LIN {X 0,Y 199.177,Z 547.457,A -85,B 0,C 180,E1 21373.917,E2 21373.917} C_VEL
LIN {X 0,Y 215.115,Z 524.972,A -85,B 0,C 180,E1 21379.948,E2 21379.948} C_VEL
LIN {X 0,Y 227.752,Z 503.08,A -85,B 0,C 180,E1 21383.961,E2 21383.961} C_VEL
LIN {X 0,Y 227.913,Z 485.066,A -85,B 0,C 180,E1 21390.32,E2 21390.32} C_VEL
LIN {X 0,Y 225.682,Z 468.338,A -85,B 0,C 180,E1 21397.834,E2 21397.834} C_VEL
LIN {X 0,Y 223.444,Z 458.289,A -85,B 0,C 180,E1 21404.278,E2 21404.278} C_VEL
LIN {X 0,Y 222.036,Z 452.317,A -85,B 0,C 180,E1 21410.188,E2 21410.188} C_VEL
LIN {X 0,Y 221.908,Z 448.763,A -85,B 0,C 180,E1 21416.091,E2 21416.091} C_VEL
LIN {X 0,Y 222.152,Z 448.898,A -85,B 0,C 180,E1 21420.003,E2 21420.003} C_VEL
LIN {X 0,Y 223.226,Z 453.842,A -85,B 0,C 180,E1 21426.819,E2 21426.819} C_VEL
LIN {X 0,Y 226.174,Z 464.487,A -85,B 0,C 180,E1 21434.54,E2 21434.54} C_VEL
LIN {X 0,Y 229.513,Z 478.492,A -85,B 0,C 180,E1 21441.276,E2 21441.276} C_VEL
LIN {X 0,Y 231.824,Z 496.438,A -85,B 0,C 180,E1 21447.624,E2 21447.624} C_VEL
LIN {X 0,Y 231.749,Z 502.452,A -85,B 0,C 180,E1 21449.308,E2 21449.308} C_VEL
LIN {X 0,Y 215.555,Z 532.804,A -85,B 0,C 180,E1 21453.677,E2 21453.677} C_VEL
LIN {X 0,Y 197.818,Z 560.36,A -85,B 0,C 180,E1 21460.055,E2 21460.055} C_VEL
LIN {X 0,Y 181.866,Z 582.088,A -85,B 0,C 180,E1 21468.235,E2 21468.235} C_VEL
LIN {X 0,Y 169.045,Z 599.486,A -85,B 0,C 180,E1 21478.996,E2 21478.996} C_VEL
LIN {X 0,Y 162.169,Z 610.738,A -85,B 0,C 180,E1 21490.92,E2 21490.92} C_VEL
LIN {X 0,Y 160.605,Z 615.153,A -85,B 0,C 180,E1 21499.125,E2 21499.125} C_VEL
LIN {X 0,Y 160.77,Z 617.402,A -85,B 0,C 180,E1 21509.992,E2 21509.992} C_VEL
LIN {X 0,Y 160.648,Z 615.185,A -85,B 0,C 180,E1 21520.856,E2 21520.856} C_VEL
LIN {X 0,Y 161.483,Z 612.541,A -85,B 0,C 180,E1 21526.327,E2 21526.327} C_VEL
LIN {X 0,Y 170.904,Z 608.235,A -85,B 0,C 180,E1 21542.098,E2 21542.098} C_VEL
LIN {X 0,Y 192.339,Z 598.523,A -85,B 0,C 180,E1 21555.096,E2 21555.096} C_VEL
LIN {X 0,Y 202.815,Z 593.917,A -85,B 0,C 180,E1 21558.952,E2 21558.952} C_VEL
LIN {X 0,Y 200.293,Z 594.401,A -85,B 0,C 180,E1 21560.543,E2 21560.543} C_VEL
LIN {X 0,Y 180.77,Z 597.692,A -85,B 0,C 180,E1 21569.832,E2 21569.832} C_VEL
LIN {X 0,Y 169.639,Z 596.938,A -85,B 0,C 180,E1 21579.082,E2 21579.082} C_VEL
LIN {X 0,Y 162.377,Z 590.884,A -85,B 0,C 180,E1 21591.957,E2 21591.957} C_VEL
LIN {X 0,Y 160.932,Z 581.155,A -85,B 0,C 180,E1 21602.692,E2 21602.692} C_VEL
LIN {X 0,Y 162.1,Z 567.404,A -85,B 0,C 180,E1 21612.606,E2 21612.606} C_VEL
LIN {X 0,Y 165.856,Z 547.555,A -85,B 0,C 180,E1 21622.423,E2 21622.423} C_VEL
LIN {X 0,Y 167.025,Z 542.957,A -85,B 0,C 180,E1 21624.287,E2 21624.287} C_VEL
LIN {X 0,Y 181.526,Z 540.142,A -85,B 0,C 180,E1 21632.822,E2 21632.822} C_VEL
LIN {X 0,Y 209.455,Z 532.398,A -85,B 0,C 180,E1 21641.296,E2 21641.296} C_VEL
LIN {X 0,Y 209.889,Z 533.058,A -85,B 0,C 180,E1 21641.79,E2 21641.79} C_VEL
LIN {X 0,Y 192.98,Z 555.356,A -85,B 0,C 180,E1 21648.886,E2 21648.886} C_VEL
LIN {X 0,Y 182.434,Z 564.426,A -85,B 0,C 180,E1 21652.185,E2 21652.185} C_VEL
LIN {X 0,Y 172.325,Z 572.215,A -85,B 0,C 180,E1 21656.038,E2 21656.038} C_VEL
LIN {X 0,Y 160.406,Z 584.48,A -85,B 0,C 180,E1 21667.828,E2 21667.828} C_VEL
LIN {X 0,Y 155.075,Z 590.148,A -85,B 0,C 180,E1 21678.749,E2 21678.749} C_VEL
LIN {X 0,Y 153.359,Z 591.986,A -85,B 0,C 180,E1 21690.008,E2 21690.008} C_VEL
LIN {X 0,Y 156.005,Z 589.027,A -85,B 0,C 180,E1 21703.985,E2 21703.985} C_VEL
LIN {X 0,Y 163.582,Z 581.161,A -85,B 0,C 180,E1 21716.088,E2 21716.088} C_VEL
LIN {X 0,Y 176.711,Z 567.47,A -85,B 0,C 180,E1 21726.858,E2 21726.858} C_VEL
LIN {X 0,Y 193.582,Z 548.12,A -85,B 0,C 180,E1 21735.541,E2 21735.541} C_VEL
LIN {X 0,Y 211.371,Z 523.809,A -85,B 0,C 180,E1 21741.996,E2 21741.996} C_VEL
LIN {X 0,Y 221.798,Z 506.936,A -85,B 0,C 180,E1 21745.004,E2 21745.004} C_VEL
LIN {X 0,Y 222.86,Z 490.693,A -85,B 0,C 180,E1 21750.937,E2 21750.937} C_VEL
LIN {X 0,Y 221.632,Z 475.531,A -85,B 0,C 180,E1 21757.936,E2 21757.936} C_VEL
LIN {X 0,Y 219.974,Z 465.484,A -85,B 0,C 180,E1 21764.499,E2 21764.499} C_VEL
LIN {X 0,Y 218.806,Z 459.156,A -85,B 0,C 180,E1 21771.173,E2 21771.173} C_VEL
LIN {X 0,Y 218.997,Z 456.251,A -85,B 0,C 180,E1 21776.039,E2 21776.039} C_VEL
LIN {X 0,Y 219.233,Z 456.387,A -85,B 0,C 180,E1 21780.003,E2 21780.003} C_VEL
LIN {X 0,Y 220.349,Z 462.641,A -85,B 0,C 180,E1 21787.901,E2 21787.901} C_VEL
LIN {X 0,Y 223.108,Z 474.069,A -85,B 0,C 180,E1 21795.752,E2 21795.752} C_VEL
LIN {X 0,Y 225.619,Z 489.59,A -85,B 0,C 180,E1 21802.7,E2 21802.7} C_VEL
LIN {X 0,Y 226.479,Z 503.724,A -85,B 0,C 180,E1 21807.631,E2 21807.631} C_VEL
LIN {X 0,Y 209.961,Z 534.007,A -85,B 0,C 180,E1 21812.2,E2 21812.2} C_VEL
LIN {X 0,Y 191.432,Z 561.307,A -85,B 0,C 180,E1 21818.711,E2 21818.711} C_VEL
LIN {X 0,Y 174.369,Z 583.318,A -85,B 0,C 180,E1 21827.422,E2 21827.422} C_VEL
LIN {X 0,Y 160.676,Z 600.703,A -85,B 0,C 180,E1 21839.171,E2 21839.171} C_VEL
LIN {X 0,Y 154.488,Z 610.163,A -85,B 0,C 180,E1 21850.074,E2 21850.074} C_VEL
LIN {X 0,Y 152.751,Z 614.505,A -85,B 0,C 180,E1 21858.558,E2 21858.558} C_VEL
LIN {X 0,Y 152.874,Z 616.764,A -85,B 0,C 180,E1 21869.992,E2 21869.992} C_VEL
LIN {X 0,Y 152.815,Z 614.539,A -85,B 0,C 180,E1 21881.42,E2 21881.42} C_VEL
LIN {X 0,Y 153.758,Z 611.875,A -85,B 0,C 180,E1 21887.172,E2 21887.172} C_VEL
LIN {X 0,Y 166.907,Z 606.908,A -85,B 0,C 180,E1 21905.966,E2 21905.966} C_VEL
LIN {X 0,Y 192.972,Z 596.975,A -85,B 0,C 180,E1 21919.08,E2 21919.08} C_VEL
LIN {X 0,Y 190.683,Z 597.243,A -85,B 0,C 180,E1 21920.565,E2 21920.565} C_VEL
LIN {X 0,Y 167.495,Z 598.655,A -85,B 0,C 180,E1 21933.129,E2 21933.129} C_VEL
LIN {X 0,Y 156.735,Z 594.166,A -85,B 0,C 180,E1 21946.023,E2 21946.023} C_VEL
LIN {X 0,Y 153.33,Z 584.856,A -85,B 0,C 180,E1 21958.582,E2 21958.582} C_VEL
LIN {X 0,Y 153.787,Z 570.942,A -85,B 0,C 180,E1 21970.171,E2 21970.171} C_VEL
LIN {X 0,Y 157.168,Z 550.928,A -85,B 0,C 180,E1 21981.171,E2 21981.171} C_VEL
LIN {X 0,Y 157.889,Z 548.939,A -85,B 0,C 180,E1 21982.549,E2 21982.549} C_VEL
LIN {X 0,Y 176.43,Z 545.25,A -85,B 0,C 180,E1 21993.896,E2 21993.896} C_VEL
LIN {X 0,Y 200.361,Z 539.066,A -85,B 0,C 180,E1 22001.377,E2 22001.377} C_VEL
LIN {X 0,Y 185.688,Z 557.62,A -85,B 0,C 180,E1 22007.987,E2 22007.987} C_VEL
LIN {X 0,Y 172.325,Z 572.215,A -85,B 0,C 180,E1 22016.038,E2 22016.038} C_VEL
LIN {X 0,Y 162.691,Z 578.921,A -85,B 0,C 180,E1 22020.5,E2 22020.5} C_VEL
LIN {X 0,Y 153.884,Z 584.343,A -85,B 0,C 180,E1 22025.631,E2 22025.631} C_VEL
LIN {X 0,Y 147.346,Z 590.785,A -85,B 0,C 180,E1 22038.151,E2 22038.151} C_VEL
LIN {X 0,Y 145.513,Z 592.621,A -85,B 0,C 180,E1 22050.009,E2 22050.009} C_VEL
LIN {X 0,Y 148.359,Z 589.665,A -85,B 0,C 180,E1 22064.721,E2 22064.721} C_VEL
LIN {X 0,Y 156.51,Z 581.805,A -85,B 0,C 180,E1 22077.362,E2 22077.362} C_VEL
LIN {X 0,Y 170.435,Z 568.125,A -85,B 0,C 180,E1 22088.457,E2 22088.457} C_VEL
LIN {X 0,Y 188.147,Z 548.795,A -85,B 0,C 180,E1 22097.254,E2 22097.254} C_VEL
LIN {X 0,Y 206.616,Z 524.515,A -85,B 0,C 180,E1 22103.717,E2 22103.717} C_VEL
LIN {X 0,Y 216.312,Z 509.416,A -85,B 0,C 180,E1 22106.433,E2 22106.433} C_VEL
LIN {X 0,Y 217.663,Z 493.427,A -85,B 0,C 180,E1 22112.765,E2 22112.765} C_VEL
LIN {X 0,Y 217.088,Z 479.857,A -85,B 0,C 180,E1 22119.596,E2 22119.596} C_VEL
LIN {X 0,Y 215.907,Z 470.26,A -85,B 0,C 180,E1 22126.727,E2 22126.727} C_VEL
LIN {X 0,Y 215.801,Z 463.629,A -85,B 0,C 180,E1 22135.98,E2 22135.98} C_VEL
LIN {X 0,Y 216.058,Z 463.769,A -85,B 0,C 180,E1 22140.003,E2 22140.003} C_VEL
LIN {X 0,Y 217.033,Z 470.12,A -85,B 0,C 180,E1 22148.022,E2 22148.022} C_VEL
LIN {X 0,Y 219.239,Z 482.003,A -85,B 0,C 180,E1 22156.037,E2 22156.037} C_VEL
LIN {X 0,Y 220.857,Z 498.201,A -85,B 0,C 180,E1 22163.215,E2 22163.215} C_VEL
LIN {X 0,Y 220.919,Z 507.282,A -85,B 0,C 180,E1 22166.459,E2 22166.459} C_VEL
LIN {X 0,Y 203.853,Z 536.285,A -85,B 0,C 180,E1 22170.849,E2 22170.849} C_VEL
LIN {X 0,Y 185.494,Z 561.798,A -85,B 0,C 180,E1 22177.13,E2 22177.13} C_VEL
LIN {X 0,Y 168.145,Z 582.98,A -85,B 0,C 180,E1 22185.713,E2 22185.713} C_VEL
LIN {X 0,Y 153.562,Z 600.243,A -85,B 0,C 180,E1 22197.81,E2 22197.81} C_VEL
LIN {X 0,Y 146.69,Z 609.895,A -85,B 0,C 180,E1 22209.67,E2 22209.67} C_VEL
LIN {X 0,Y 144.904,Z 613.856,A -85,B 0,C 180,E1 22217.93,E2 22217.93} C_VEL
LIN {X 0,Y 144.977,Z 616.125,A -85,B 0,C 180,E1 22229.991,E2 22229.991} C_VEL
LIN {X 0,Y 144.97,Z 613.892,A -85,B 0,C 180,E1 22242.047,E2 22242.047} C_VEL
LIN {X 0,Y 146.908,Z 610.149,A -85,B 0,C 180,E1 22250.483,E2 22250.483} C_VEL
LIN {X 0,Y 160.601,Z 606.569,A -85,B 0,C 180,E1 22267.777,E2 22267.777} C_VEL
LIN {X 0,Y 182.654,Z 599.585,A -85,B 0,C 180,E1 22279.069,E2 22279.069} C_VEL
LIN {X 0,Y 181.918,Z 599.433,A -85,B 0,C 180,E1 22280.198,E2 22280.198} C_VEL
LIN {X 0,Y 160.523,Z 599.431,A -85,B 0,C 180,E1 22291.861,E2 22291.861} C_VEL
LIN {X 0,Y 148.97,Z 594.046,A -85,B 0,C 180,E1 22305.479,E2 22305.479} C_VEL
LIN {X 0,Y 145.459,Z 584.242,A -85,B 0,C 180,E1 22318.505,E2 22318.505} C_VEL
LIN {X 0,Y 145.985,Z 569.601,A -85,B 0,C 180,E1 22330.721,E2 22330.721} C_VEL
LIN {X 0,Y 148.737,Z 554.448,A -85,B 0,C 180,E1 22340.088,E2 22340.088} C_VEL
LIN {X 0,Y 171.246,Z 550.073,A -85,B 0,C 180,E1 22355.07,E2 22355.07} C_VEL
LIN {X 0,Y 190.552,Z 545.467,A -85,B 0,C 180,E1 22361.307,E2 22361.307} C_VEL
LIN {X 0,Y 175.103,Z 563.43,A -85,B 0,C 180,E1 22368.767,E2 22368.767} C_VEL
LIN {X 0,Y 160.002,Z 578.515,A -85,B 0,C 180,E1 22379.091,E2 22379.091} C_VEL
LIN {X 0,Y 153.884,Z 584.343,A -85,B 0,C 180,E1 22385.631,E2 22385.631} C_VEL
LIN {X 0,Y 146.298,Z 588.632,A -85,B 0,C 180,E1 22391.428,E2 22391.428} C_VEL
LIN {X 0,Y 139.489,Z 591.502,A -85,B 0,C 180,E1 22397.847,E2 22397.847} C_VEL
LIN {X 0,Y 137.636,Z 593.258,A -85,B 0,C 180,E1 22410.009,E2 22410.009} C_VEL
LIN {X 0,Y 140.642,Z 590.392,A -85,B 0,C 180,E1 22425.301,E2 22425.301} C_VEL
LIN {X 0,Y 149.53,Z 582.448,A -85,B 0,C 180,E1 22438.755,E2 22438.755} C_VEL
LIN {X 0,Y 164.301,Z 568.777,A -85,B 0,C 180,E1 22450.176,E2 22450.176} C_VEL
LIN {X 0,Y 182.875,Z 549.472,A -85,B 0,C 180,E1 22459.072,E2 22459.072} C_VEL
LIN {X 0,Y 202.045,Z 525.224,A -85,B 0,C 180,E1 22465.522,E2 22465.522} C_VEL
LIN {X 0,Y 210.882,Z 512.011,A -85,B 0,C 180,E1 22467.927,E2 22467.927} C_VEL
LIN {X 0,Y 212.565,Z 497.474,A -85,B 0,C 180,E1 22474.12,E2 22474.12} C_VEL
LIN {X 0,Y 212.641,Z 484.92,A -85,B 0,C 180,E1 22480.892,E2 22480.892} C_VEL
LIN {X 0,Y 212.092,Z 475.095,A -85,B 0,C 180,E1 22489.148,E2 22489.148} C_VEL
LIN {X 0,Y 212.433,Z 470.784,A -85,B 0,C 180,E1 22496.226,E2 22496.226} C_VEL
LIN {X 0,Y 212.665,Z 471.048,A -85,B 0,C 180,E1 22500.003,E2 22500.003} C_VEL
LIN {X 0,Y 213.404,Z 477.484,A -85,B 0,C 180,E1 22508.159,E2 22508.159} C_VEL
LIN {X 0,Y 214.836,Z 488.174,A -85,B 0,C 180,E1 22515.448,E2 22515.448} C_VEL
LIN {X 0,Y 215.654,Z 503.707,A -85,B 0,C 180,E1 22522.581,E2 22522.581} C_VEL
LIN {X 0,Y 214.959,Z 511.066,A -85,B 0,C 180,E1 22525.103,E2 22525.103} C_VEL
LIN {X 0,Y 196.7,Z 539.99,A -85,B 0,C 180,E1 22529.744,E2 22529.744} C_VEL
LIN {X 0,Y 176.998,Z 565.69,A -85,B 0,C 180,E1 22536.573,E2 22536.573} C_VEL
LIN {X 0,Y 158.766,Z 586.294,A -85,B 0,C 180,E1 22545.972,E2 22545.972} C_VEL
LIN {X 0,Y 144.748,Z 601.89,A -85,B 0,C 180,E1 22558.459,E2 22558.459} C_VEL
LIN {X 0,Y 138.364,Z 610.501,A -85,B 0,C 180,E1 22570.828,E2 22570.828} C_VEL
LIN {X 0,Y 136.72,Z 614.84,A -85,B 0,C 180,E1 22583.633,E2 22583.633} C_VEL
LIN {X 0,Y 137.078,Z 615.485,A -85,B 0,C 180,E1 22589.991,E2 22589.991} C_VEL
LIN {X 0,Y 137.141,Z 613.244,A -85,B 0,C 180,E1 22602.745,E2 22602.745} C_VEL
LIN {X 0,Y 140.214,Z 608.914,A -85,B 0,C 180,E1 22613.505,E2 22613.505} C_VEL
LIN {X 0,Y 158.032,Z 605.249,A -85,B 0,C 180,E1 22632.102,E2 22632.102} C_VEL
LIN {X 0,Y 171.29,Z 601.783,A -85,B 0,C 180,E1 22638.657,E2 22638.657} C_VEL
LIN {X 0,Y 172.797,Z 601.214,A -85,B 0,C 180,E1 22639.877,E2 22639.877} C_VEL
LIN {X 0,Y 153.627,Z 600.092,A -85,B 0,C 180,E1 22650.476,E2 22650.476} C_VEL
LIN {X 0,Y 140.769,Z 593.255,A -85,B 0,C 180,E1 22665.839,E2 22665.839} C_VEL
LIN {X 0,Y 137.429,Z 581.903,A -85,B 0,C 180,E1 22679.996,E2 22679.996} C_VEL
LIN {X 0,Y 138.221,Z 568.205,A -85,B 0,C 180,E1 22691.304,E2 22691.304} C_VEL
LIN {X 0,Y 139.695,Z 559.704,A -85,B 0,C 180,E1 22697.335,E2 22697.335} C_VEL
LIN {X 0,Y 161.307,Z 555.607,A -85,B 0,C 180,E1 22714.267,E2 22714.267} C_VEL
LIN {X 0,Y 180.578,Z 551.515,A -85,B 0,C 180,E1 22721.239,E2 22721.239} C_VEL
LIN {X 0,Y 177.835,Z 555.21,A -85,B 0,C 180,E1 22722.92,E2 22722.92} C_VEL
LIN {X 0,Y 160.43,Z 572.578,A -85,B 0,C 180,E1 22732.176,E2 22732.176} C_VEL
LIN {X 0,Y 146.442,Z 585.224,A -85,B 0,C 180,E1 22744.702,E2 22744.702} C_VEL
LIN {X 0,Y 139.489,Z 591.502,A -85,B 0,C 180,E1 22757.847,E2 22757.847} C_VEL
LIN {X 0,Y 133.921,Z 593.276,A -85,B 0,C 180,E1 22764.753,E2 22764.753} C_VEL
LIN {X 0,Y 129.705,Z 593.729,A -85,B 0,C 180,E1 22772.169,E2 22772.169} C_VEL
LIN {X 0,Y 133.161,Z 590.92,A -85,B 0,C 180,E1 22786.523,E2 22786.523} C_VEL
LIN {X 0,Y 142.641,Z 583.091,A -85,B 0,C 180,E1 22800.285,E2 22800.285} C_VEL
LIN {X 0,Y 158.347,Z 569.428,A -85,B 0,C 180,E1 22812.021,E2 22812.021} C_VEL
LIN {X 0,Y 177.792,Z 550.149,A -85,B 0,C 180,E1 22820.999,E2 22820.999} C_VEL
LIN {X 0,Y 197.697,Z 525.933,A -85,B 0,C 180,E1 22827.402,E2 22827.402} C_VEL
LIN {X 0,Y 205.54,Z 514.4,A -85,B 0,C 180,E1 22829.642,E2 22829.642} C_VEL
LIN {X 0,Y 207.567,Z 501.324,A -85,B 0,C 180,E1 22835.594,E2 22835.594} C_VEL
LIN {X 0,Y 208.143,Z 490.302,A -85,B 0,C 180,E1 22841.997,E2 22841.997} C_VEL
LIN {X 0,Y 208.188,Z 481.816,A -85,B 0,C 180,E1 22849.528,E2 22849.528} C_VEL
LIN {X 0,Y 208.744,Z 478.088,A -85,B 0,C 180,E1 22855.844,E2 22855.844} C_VEL
LIN {X 0,Y 209.065,Z 478.207,A -85,B 0,C 180,E1 22860.003,E2 22860.003} C_VEL
LIN {X 0,Y 209.479,Z 484.8,A -85,B 0,C 180,E1 22868.313,E2 22868.313} C_VEL
LIN {X 0,Y 210.352,Z 495.679,A -85,B 0,C 180,E1 22875.66,E2 22875.66} C_VEL
LIN {X 0,Y 210.201,Z 511.241,A -85,B 0,C 180,E1 22882.779,E2 22882.779} C_VEL
LIN {X 0,Y 209.033,Z 514.658,A -85,B 0,C 180,E1 22883.673,E2 22883.673} C_VEL
LIN {X 0,Y 189.597,Z 543.646,A -85,B 0,C 180,E1 22888.542,E2 22888.542} C_VEL
LIN {X 0,Y 169.651,Z 567.882,A -85,B 0,C 180,E1 22895.446,E2 22895.446} C_VEL
LIN {X 0,Y 150.704,Z 587.978,A -85,B 0,C 180,E1 22905.303,E2 22905.303} C_VEL
LIN {X 0,Y 136.66,Z 602.512,A -85,B 0,C 180,E1 22918.239,E2 22918.239} C_VEL
LIN {X 0,Y 129.844,Z 611.31,A -85,B 0,C 180,E1 22933.042,E2 22933.042} C_VEL
LIN {X 0,Y 128.808,Z 614.195,A -85,B 0,C 180,E1 22943.24,E2 22943.24} C_VEL
LIN {X 0,Y 129.204,Z 614.848,A -85,B 0,C 180,E1 22949.99,E2 22949.99} C_VEL
LIN {X 0,Y 129.329,Z 612.596,A -85,B 0,C 180,E1 22963.529,E2 22963.529} C_VEL
LIN {X 0,Y 132.998,Z 607.618,A -85,B 0,C 180,E1 22975.033,E2 22975.033} C_VEL
LIN {X 0,Y 152.158,Z 604.861,A -85,B 0,C 180,E1 22994.134,E2 22994.134} C_VEL
LIN {X 0,Y 162.831,Z 602.613,A -85,B 0,C 180,E1 22999.392,E2 22999.392} C_VEL
LIN {X 0,Y 140.546,Z 598.526,A -85,B 0,C 180,E1 23014.473,E2 23014.473} C_VEL
LIN {X 0,Y 131.264,Z 589.48,A -85,B 0,C 180,E1 23030.033,E2 23030.033} C_VEL
LIN {X 0,Y 129.471,Z 577.442,A -85,B 0,C 180,E1 23043.347,E2 23043.347} C_VEL
LIN {X 0,Y 130.723,Z 564.733,A -85,B 0,C 180,E1 23053.388,E2 23053.388} C_VEL
LIN {X 0,Y 155.911,Z 559.992,A -85,B 0,C 180,E1 23075.629,E2 23075.629} C_VEL
LIN {X 0,Y 170.564,Z 557.157,A -85,B 0,C 180,E1 23081.17,E2 23081.17} C_VEL
LIN {X 0,Y 169.026,Z 559.373,A -85,B 0,C 180,E1 23082.491,E2 23082.491} C_VEL
LIN {X 0,Y 150.549,Z 576.474,A -85,B 0,C 180,E1 23092.9,E2 23092.9} C_VEL
LIN {X 0,Y 138.702,Z 586.399,A -85,B 0,C 180,E1 23104.123,E2 23104.123} C_VEL
LIN {X 0,Y 131.729,Z 592.174,A -85,B 0,C 180,E1 23117.29,E2 23117.29} C_VEL
LIN {X 0,Y 129.705,Z 593.729,A -85,B 0,C 180,E1 23132.169,E2 23132.169} C_VEL
LIN {X 0,Y 128.791,Z 593.589,A -85,B 0,C 180,E1 23136.027,E2 23136.027} C_VEL
LIN {X 0,Y 125.412,Z 591.794,A -85,B 0,C 180,E1 23146.863,E2 23146.863} C_VEL
LIN {X 0,Y 125.743,Z 591.444,A -85,B 0,C 180,E1 23147.846,E2 23147.846} C_VEL
LIN {X 0,Y 137.412,Z 582.478,A -85,B 0,C 180,E1 23163.438,E2 23163.438} C_VEL
LIN {X 0,Y 154.74,Z 568.203,A -85,B 0,C 180,E1 23175.191,E2 23175.191} C_VEL
LIN {X 0,Y 174.256,Z 549.401,A -85,B 0,C 180,E1 23183.491,E2 23183.491} C_VEL
LIN {X 0,Y 194.63,Z 525.25,A -85,B 0,C 180,E1 23189.649,E2 23189.649} C_VEL
LIN {X 0,Y 199.715,Z 518.278,A -85,B 0,C 180,E1 23190.894,E2 23190.894} C_VEL
LIN {X 0,Y 202.28,Z 507.251,A -85,B 0,C 180,E1 23196.031,E2 23196.031} C_VEL
LIN {X 0,Y 203.544,Z 496.214,A -85,B 0,C 180,E1 23202.695,E2 23202.695} C_VEL
LIN {X 0,Y 204.115,Z 488.415,A -85,B 0,C 180,E1 23209.962,E2 23209.962} C_VEL
LIN {X 0,Y 204.853,Z 485.115,A -85,B 0,C 180,E1 23215.765,E2 23215.765} C_VEL
LIN {X 0,Y 205.181,Z 485.204,A -85,B 0,C 180,E1 23220.003,E2 23220.003} C_VEL
LIN {X 0,Y 205.276,Z 490.817,A -85,B 0,C 180,E1 23227.418,E2 23227.418} C_VEL
LIN {X 0,Y 205.573,Z 501.41,A -85,B 0,C 180,E1 23234.942,E2 23234.942} C_VEL
LIN {X 0,Y 204.756,Z 515.453,A -85,B 0,C 180,E1 23241.699,E2 23241.699} C_VEL
LIN {X 0,Y 184.073,Z 545.131,A -85,B 0,C 180,E1 23246.834,E2 23246.834} C_VEL
LIN {X 0,Y 162.766,Z 569.644,A -85,B 0,C 180,E1 23254.057,E2 23254.057} C_VEL
LIN {X 0,Y 142.99,Z 589.205,A -85,B 0,C 180,E1 23264.371,E2 23264.371} C_VEL
LIN {X 0,Y 128.55,Z 603.092,A -85,B 0,C 180,E1 23277.985,E2 23277.985} C_VEL
LIN {X 0,Y 122.174,Z 610.659,A -85,B 0,C 180,E1 23291.942,E2 23291.942} C_VEL
LIN {X 0,Y 120.899,Z 613.55,A -85,B 0,C 180,E1 23302.796,E2 23302.796} C_VEL
LIN {X 0,Y 121.14,Z 614.157,A -85,B 0,C 180,E1 23310.976,E2 23310.976} C_VEL
LIN {X 0,Y 121.548,Z 611.947,A -85,B 0,C 180,E1 23324.414,E2 23324.414} C_VEL
LIN {X 0,Y 126.873,Z 606.301,A -85,B 0,C 180,E1 23338.498,E2 23338.498} C_VEL
LIN {X 0,Y 146.519,Z 604.336,A -85,B 0,C 180,E1 23356.314,E2 23356.314} C_VEL
LIN {X 0,Y 152.448,Z 603.18,A -85,B 0,C 180,E1 23359.793,E2 23359.793} C_VEL
LIN {X 0,Y 133.459,Z 598.549,A -85,B 0,C 180,E1 23373.011,E2 23373.011} C_VEL
LIN {X 0,Y 123.623,Z 588.993,A -85,B 0,C 180,E1 23389.117,E2 23389.117} C_VEL
LIN {X 0,Y 121.644,Z 577.998,A -85,B 0,C 180,E1 23401.766,E2 23401.766} C_VEL
LIN {X 0,Y 122.248,Z 569.693,A -85,B 0,C 180,E1 23409.799,E2 23409.799} C_VEL
LIN {X 0,Y 150.501,Z 564.18,A -85,B 0,C 180,E1 23437.12,E2 23437.12} C_VEL
LIN {X 0,Y 160.838,Z 562.349,A -85,B 0,C 180,E1 23441.21,E2 23441.21} C_VEL
LIN {X 0,Y 156.837,Z 566.466,A -85,B 0,C 180,E1 23443.654,E2 23443.654} C_VEL
LIN {X 0,Y 139.17,Z 581.176,A -85,B 0,C 180,E1 23454.907,E2 23454.907} C_VEL
LIN {X 0,Y 127.249,Z 590.356,A -85,B 0,C 180,E1 23469.1,E2 23469.1} C_VEL
LIN {X 0,Y 122.336,Z 594.051,A -85,B 0,C 180,E1 23482.902,E2 23482.902} C_VEL
LIN {X 0,Y 122.363,Z 594.017,A -85,B 0,C 180,E1 23497.118,E2 23497.118} C_VEL
LIN {X 0,Y 125.743,Z 591.444,A -85,B 0,C 180,E1 23507.846,E2 23507.846} C_VEL
LIN {X 0,Y 126.247,Z 588.646,A -85,B 0,C 180,E1 23515.709,E2 23515.709} C_VEL
LIN {X 0,Y 128.708,Z 584.718,A -85,B 0,C 180,E1 23523.345,E2 23523.345} C_VEL
LIN {X 0,Y 146.969,Z 570.732,A -85,B 0,C 180,E1 23536.156,E2 23536.156} C_VEL
LIN {X 0,Y 168.311,Z 551.494,A -85,B 0,C 180,E1 23545.176,E2 23545.176} C_VEL
LIN {X 0,Y 189.679,Z 527.345,A -85,B 0,C 180,E1 23551.413,E2 23551.413} C_VEL
LIN {X 0,Y 194.77,Z 520.67,A -85,B 0,C 180,E1 23552.63,E2 23552.63} C_VEL
LIN {X 0,Y 197.791,Z 508.325,A -85,B 0,C 180,E1 23559.204,E2 23559.204} C_VEL
LIN {X 0,Y 199.196,Z 499.247,A -85,B 0,C 180,E1 23565.739,E2 23565.739} C_VEL
LIN {X 0,Y 199.973,Z 494.357,A -85,B 0,C 180,E1 23571.294,E2 23571.294} C_VEL
LIN {X 0,Y 200.695,Z 491.986,A -85,B 0,C 180,E1 23575.677,E2 23575.677} C_VEL
LIN {X 0,Y 201.068,Z 492.055,A -85,B 0,C 180,E1 23580.003,E2 23580.003} C_VEL
LIN {X 0,Y 200.949,Z 497.876,A -85,B 0,C 180,E1 23587.579,E2 23587.579} C_VEL
LIN {X 0,Y 200.666,Z 507.493,A -85,B 0,C 180,E1 23594.476,E2 23594.476} C_VEL
LIN {X 0,Y 199.104,Z 519.316,A -85,B 0,C 180,E1 23600.285,E2 23600.285} C_VEL
LIN {X 0,Y 178.301,Z 547.105,A -85,B 0,C 180,E1 23605.125,E2 23605.125} C_VEL
LIN {X 0,Y 156.437,Z 570.883,A -85,B 0,C 180,E1 23612.366,E2 23612.366} C_VEL
LIN {X 0,Y 135.315,Z 590.374,A -85,B 0,C 180,E1 23623.331,E2 23623.331} C_VEL
LIN {X 0,Y 120.473,Z 603.668,A -85,B 0,C 180,E1 23637.706,E2 23637.706} C_VEL
LIN {X 0,Y 113.714,Z 611.259,A -85,B 0,C 180,E1 23654.546,E2 23654.546} C_VEL
LIN {X 0,Y 113.431,Z 613.572,A -85,B 0,C 180,E1 23669.989,E2 23669.989} C_VEL
LIN {X 0,Y 113.786,Z 611.298,A -85,B 0,C 180,E1 23685.421,E2 23685.421} C_VEL
LIN {X 0,Y 121.122,Z 604.822,A -85,B 0,C 180,E1 23702.075,E2 23702.075} C_VEL
LIN {X 0,Y 141.104,Z 603.54,A -85,B 0,C 180,E1 23718.667,E2 23718.667} C_VEL
LIN {X 0,Y 142.023,Z 603.118,A -85,B 0,C 180,E1 23720.235,E2 23720.235} C_VEL
LIN {X 0,Y 123.495,Z 596.805,A -85,B 0,C 180,E1 23734.587,E2 23734.587} C_VEL
LIN {X 0,Y 114.825,Z 585.036,A -85,B 0,C 180,E1 23752.419,E2 23752.419} C_VEL
LIN {X 0,Y 113.823,Z 574.715,A -85,B 0,C 180,E1 23763.782,E2 23763.782} C_VEL
LIN {X 0,Y 148.775,Z 567.469,A -85,B 0,C 180,E1 23800.305,E2 23800.305} C_VEL
LIN {X 0,Y 150.456,Z 567.18,A -85,B 0,C 180,E1 23800.96,E2 23800.96} C_VEL
LIN {X 0,Y 149.132,Z 569.101,A -85,B 0,C 180,E1 23802.64,E2 23802.64} C_VEL
LIN {X 0,Y 130.769,Z 583.28,A -85,B 0,C 180,E1 23814.642,E2 23814.642} C_VEL
LIN {X 0,Y 119.894,Z 590.996,A -85,B 0,C 180,E1 23827.751,E2 23827.751} C_VEL
LIN {X 0,Y 114.533,Z 594.687,A -85,B 0,C 180,E1 23842.416,E2 23842.416} C_VEL
LIN {X 0,Y 114.56,Z 594.654,A -85,B 0,C 180,E1 23857.605,E2 23857.605} C_VEL
LIN {X 0,Y 119.939,Z 590.902,A -85,B 0,C 180,E1 23872.263,E2 23872.263} C_VEL
LIN {X 0,Y 128.708,Z 584.718,A -85,B 0,C 180,E1 23883.345,E2 23883.345} C_VEL
LIN {X 0,Y 132.962,Z 579.725,A -85,B 0,C 180,E1 23890.477,E2 23890.477} C_VEL
LIN {X 0,Y 138.748,Z 573.608,A -85,B 0,C 180,E1 23896.984,E2 23896.984} C_VEL
LIN {X 0,Y 161.131,Z 554.747,A -85,B 0,C 180,E1 23906.52,E2 23906.52} C_VEL
LIN {X 0,Y 182.659,Z 532.195,A -85,B 0,C 180,E1 23912.74,E2 23912.74} C_VEL
LIN {X 0,Y 189.708,Z 523.378,A -85,B 0,C 180,E1 23914.455,E2 23914.455} C_VEL
LIN {X 0,Y 193.301,Z 510.949,A -85,B 0,C 180,E1 23921.746,E2 23921.746} C_VEL
LIN {X 0,Y 194.901,Z 503.458,A -85,B 0,C 180,E1 23928.182,E2 23928.182} C_VEL
LIN {X 0,Y 196.319,Z 498.748,A -85,B 0,C 180,E1 23935.58,E2 23935.58} C_VEL
LIN {X 0,Y 196.748,Z 498.793,A -85,B 0,C 180,E1 23940.003,E2 23940.003} C_VEL
LIN {X 0,Y 196.276,Z 504.821,A -85,B 0,C 180,E1 23947.76,E2 23947.76} C_VEL
LIN {X 0,Y 195.363,Z 514.44,A -85,B 0,C 180,E1 23954.59,E2 23954.59} C_VEL
LIN {X 0,Y 194.339,Z 521.071,A -85,B 0,C 180,E1 23958.159,E2 23958.159} C_VEL
LIN {X 0,Y 182.411,Z 537.524,A -85,B 0,C 180,E1 23960.961,E2 23960.961} C_VEL
LIN {X 0,Y 159.54,Z 563.045,A -85,B 0,C 180,E1 23967.156,E2 23967.156} C_VEL
LIN {X 0,Y 136.783,Z 583.896,A -85,B 0,C 180,E1 23976.621,E2 23976.621} C_VEL
LIN {X 0,Y 118.051,Z 599.351,A -85,B 0,C 180,E1 23990.312,E2 23990.312} C_VEL
LIN {X 0,Y 108.316,Z 607.874,A -85,B 0,C 180,E1 24005.196,E2 24005.196} C_VEL
LIN {X 0,Y 105.103,Z 612.26,A -85,B 0,C 180,E1 24021.706,E2 24021.706} C_VEL
LIN {X 0,Y 105.521,Z 612.932,A -85,B 0,C 180,E1 24029.988,E2 24029.988} C_VEL
LIN {X 0,Y 106.06,Z 610.649,A -85,B 0,C 180,E1 24046.575,E2 24046.575} C_VEL
LIN {X 0,Y 114.459,Z 603.224,A -85,B 0,C 180,E1 24064.19,E2 24064.19} C_VEL
LIN {X 0,Y 131.203,Z 602.977,A -85,B 0,C 180,E1 24078.577,E2 24078.577} C_VEL
LIN {X 0,Y 132.476,Z 602.664,A -85,B 0,C 180,E1 24080.064,E2 24080.064} C_VEL
LIN {X 0,Y 112.457,Z 593.218,A -85,B 0,C 180,E1 24098.266,E2 24098.266} C_VEL
LIN {X 0,Y 106.232,Z 579.517,A -85,B 0,C 180,E1 24117.953,E2 24117.953} C_VEL
LIN {X 0,Y 141.459,Z 571.618,A -85,B 0,C 180,E1 24161.496,E2 24161.496} C_VEL
LIN {X 0,Y 122.614,Z 585.15,A -85,B 0,C 180,E1 24174.105,E2 24174.105} C_VEL
LIN {X 0,Y 110.578,Z 592.913,A -85,B 0,C 180,E1 24189.997,E2 24189.997} C_VEL
LIN {X 0,Y 106.161,Z 595.805,A -85,B 0,C 180,E1 24210.012,E2 24210.012} C_VEL
LIN {X 0,Y 110.658,Z 592.837,A -85,B 0,C 180,E1 24230.013,E2 24230.013} C_VEL
LIN {X 0,Y 122.717,Z 585.018,A -85,B 0,C 180,E1 24245.887,E2 24245.887} C_VEL
LIN {X 0,Y 138.748,Z 573.608,A -85,B 0,C 180,E1 24256.984,E2 24256.984} C_VEL
LIN {X 0,Y 145.791,Z 566.543,A -85,B 0,C 180,E1 24262.806,E2 24262.806} C_VEL
LIN {X 0,Y 153.721,Z 558.273,A -85,B 0,C 180,E1 24267.879,E2 24267.879} C_VEL
LIN {X 0,Y 176.359,Z 536.014,A -85,B 0,C 180,E1 24274.31,E2 24274.31} C_VEL
LIN {X 0,Y 184.875,Z 525.825,A -85,B 0,C 180,E1 24276.53,E2 24276.53} C_VEL
LIN {X 0,Y 188.21,Z 516.071,A -85,B 0,C 180,E1 24282.723,E2 24282.723} C_VEL
LIN {X 0,Y 190.065,Z 509.68,A -85,B 0,C 180,E1 24288.517,E2 24288.517} C_VEL
LIN {X 0,Y 191.729,Z 505.39,A -85,B 0,C 180,E1 24295.474,E2 24295.474} C_VEL
LIN {X 0,Y 192.242,Z 505.382,A -85,B 0,C 180,E1 24300.003,E2 24300.003} C_VEL
LIN {X 0,Y 191.517,Z 510.375,A -85,B 0,C 180,E1 24306.813,E2 24306.813} C_VEL
LIN {X 0,Y 190.084,Z 519.74,A -85,B 0,C 180,E1 24313.827,E2 24313.827} C_VEL
LIN {X 0,Y 188.764,Z 525.25,A -85,B 0,C 180,E1 24316.758,E2 24316.758} C_VEL
LIN {X 0,Y 166.131,Z 552.093,A -85,B 0,C 180,E1 24321.679,E2 24321.679} C_VEL
LIN {X 0,Y 141.851,Z 575.224,A -85,B 0,C 180,E1 24329.456,E2 24329.456} C_VEL
LIN {X 0,Y 120.113,Z 592.498,A -85,B 0,C 180,E1 24340.848,E2 24340.848} C_VEL
LIN {X 0,Y 104.291,Z 604.464,A -85,B 0,C 180,E1 24357.004,E2 24357.004} C_VEL
LIN {X 0,Y 98.294,Z 609.957,A -85,B 0,C 180,E1 24372.045,E2 24372.045} C_VEL
LIN {X 0,Y 97.605,Z 612.292,A -85,B 0,C 180,E1 24389.987,E2 24389.987} C_VEL
LIN {X 0,Y 98.385,Z 609.999,A -85,B 0,C 180,E1 24407.91,E2 24407.91} C_VEL
LIN {X 0,Y 109.588,Z 601.533,A -85,B 0,C 180,E1 24428.423,E2 24428.423} C_VEL
LIN {X 0,Y 121.353,Z 601.851,A -85,B 0,C 180,E1 24438.447,E2 24438.447} C_VEL
LIN {X 0,Y 122.254,Z 601.481,A -85,B 0,C 180,E1 24440.295,E2 24440.295} C_VEL
LIN {X 0,Y 104.061,Z 591.15,A -85,B 0,C 180,E1 24458.666,E2 24458.666} C_VEL
LIN {X 0,Y 99.646,Z 584.49,A -85,B 0,C 180,E1 24469.817,E2 24469.817} C_VEL
LIN {X 0,Y 103.957,Z 579.95,A -85,B 0,C 180,E1 24496.927,E2 24496.927} C_VEL
LIN {X 0,Y 130.166,Z 575.774,A -85,B 0,C 180,E1 24520.557,E2 24520.557} C_VEL
LIN {X 0,Y 131.081,Z 576.037,A -85,B 0,C 180,E1 24521.707,E2 24521.707} C_VEL
LIN {X 0,Y 112.663,Z 587.997,A -85,B 0,C 180,E1 24535.225,E2 24535.225} C_VEL
LIN {X 0,Y 101.458,Z 594.611,A -85,B 0,C 180,E1 24552.65,E2 24552.65} C_VEL
LIN {X 0,Y 98.304,Z 596.441,A -85,B 0,C 180,E1 24570.013,E2 24570.013} C_VEL
LIN {X 0,Y 103.258,Z 593.477,A -85,B 0,C 180,E1 24591.516,E2 24591.516} C_VEL
LIN {X 0,Y 116.38,Z 585.661,A -85,B 0,C 180,E1 24608.177,E2 24608.177} C_VEL
LIN {X 0,Y 136.479,Z 572.038,A -85,B 0,C 180,E1 24620.956,E2 24620.956} C_VEL
LIN {X 0,Y 153.721,Z 558.273,A -85,B 0,C 180,E1 24627.879,E2 24627.879} C_VEL
LIN {X 0,Y 162.316,Z 549.148,A -85,B 0,C 180,E1 24632.342,E2 24632.342} C_VEL
LIN {X 0,Y 169.739,Z 540.345,A -85,B 0,C 180,E1 24635.859,E2 24635.859} C_VEL
LIN {X 0,Y 171.051,Z 538.908,A -85,B 0,C 180,E1 24636.196,E2 24636.196} C_VEL
LIN {X 0,Y 179.579,Z 529.464,A -85,B 0,C 180,E1 24638.044,E2 24638.044} C_VEL
LIN {X 0,Y 183.541,Z 519.915,A -85,B 0,C 180,E1 24644.734,E2 24644.734} C_VEL
LIN {X 0,Y 185.756,Z 513.907,A -85,B 0,C 180,E1 24651.472,E2 24651.472} C_VEL
LIN {X 0,Y 186.899,Z 511.864,A -85,B 0,C 180,E1 24655.357,E2 24655.357} C_VEL
LIN {X 0,Y 187.452,Z 511.783,A -85,B 0,C 180,E1 24660.003,E2 24660.003} C_VEL
LIN {X 0,Y 186.336,Z 517.407,A -85,B 0,C 180,E1 24667.337,E2 24667.337} C_VEL
LIN {X 0,Y 184.501,Z 525.76,A -85,B 0,C 180,E1 24673.542,E2 24673.542} C_VEL
LIN {X 0,Y 183.51,Z 528.397,A -85,B 0,C 180,E1 24674.907,E2 24674.907} C_VEL
LIN {X 0,Y 159.169,Z 555.612,A -85,B 0,C 180,E1 24680.049,E2 24680.049} C_VEL
LIN {X 0,Y 133.326,Z 578.257,A -85,B 0,C 180,E1 24688.335,E2 24688.335} C_VEL
LIN {X 0,Y 110.372,Z 595.026,A -85,B 0,C 180,E1 24701.008,E2 24701.008} C_VEL
LIN {X 0,Y 96.191,Z 604.826,A -85,B 0,C 180,E1 24716.558,E2 24716.558} C_VEL
LIN {X 0,Y 90.687,Z 609.307,A -85,B 0,C 180,E1 24730.481,E2 24730.481} C_VEL
LIN {X 0,Y 89.686,Z 611.651,A -85,B 0,C 180,E1 24749.986,E2 24749.986} C_VEL
LIN {X 0,Y 90.782,Z 609.351,A -85,B 0,C 180,E1 24769.468,E2 24769.468} C_VEL
LIN {X 0,Y 103.394,Z 600.651,A -85,B 0,C 180,E1 24791.2,E2 24791.2} C_VEL
LIN {X 0,Y 108.277,Z 599.951,A -85,B 0,C 180,E1 24795.639,E2 24795.639} C_VEL
LIN {X 0,Y 112.601,Z 600.18,A -85,B 0,C 180,E1 24798.957,E2 24798.957} C_VEL
LIN {X 0,Y 110.396,Z 598.904,A -85,B 0,C 180,E1 24801.888,E2 24801.888} C_VEL
LIN {X 0,Y 95.564,Z 589.617,A -85,B 0,C 180,E1 24819.112,E2 24819.112} C_VEL
LIN {X 0,Y 93.303,Z 584.487,A -85,B 0,C 180,E1 24849.332,E2 24849.332} C_VEL
LIN {X 0,Y 121.327,Z 579.691,A -85,B 0,C 180,E1 24881.539,E2 24881.539} C_VEL
LIN {X 0,Y 104.51,Z 589.598,A -85,B 0,C 180,E1 24894.604,E2 24894.604} C_VEL
LIN {X 0,Y 93.947,Z 595.25,A -85,B 0,C 180,E1 24911.213,E2 24911.213} C_VEL
LIN {X 0,Y 90.44,Z 597.077,A -85,B 0,C 180,E1 24930.014,E2 24930.014} C_VEL
LIN {X 0,Y 95.952,Z 594.116,A -85,B 0,C 180,E1 24953.246,E2 24953.246} C_VEL
LIN {X 0,Y 110.034,Z 586.423,A -85,B 0,C 180,E1 24970.542,E2 24970.542} C_VEL
LIN {X 0,Y 131.632,Z 572.69,A -85,B 0,C 180,E1 24983.635,E2 24983.635} C_VEL
LIN {X 0,Y 156.013,Z 553.498,A -85,B 0,C 180,E1 24992.328,E2 24992.328} C_VEL
LIN {X 0,Y 171.051,Z 538.908,A -85,B 0,C 180,E1 24996.196,E2 24996.196} C_VEL
LIN {X 0,Y 174.504,Z 534.139,A -85,B 0,C 180,E1 24998.248,E2 24998.248} C_VEL
LIN {X 0,Y 176.733,Z 528.402,A -85,B 0,C 180,E1 25002.946,E2 25002.946} C_VEL
LIN {X 0,Y 179.659,Z 522.115,A -85,B 0,C 180,E1 25008.673,E2 25008.673} C_VEL
LIN {X 0,Y 181.806,Z 518.152,A -85,B 0,C 180,E1 25015.227,E2 25015.227} C_VEL
LIN {X 0,Y 182.435,Z 518.05,A -85,B 0,C 180,E1 25020.003,E2 25020.003} C_VEL
LIN {X 0,Y 181.346,Z 522.497,A -85,B 0,C 180,E1 25026.164,E2 25026.164} C_VEL
LIN {X 0,Y 179.052,Z 530.432,A -85,B 0,C 180,E1 25032.501,E2 25032.501} C_VEL
LIN {X 0,Y 172.819,Z 538.065,A -85,B 0,C 180,E1 25033.952,E2 25033.952} C_VEL
LIN {X 0,Y 146.737,Z 563.766,A -85,B 0,C 180,E1 25039.677,E2 25039.677} C_VEL
LIN {X 0,Y 120.9,Z 583.925,A -85,B 0,C 180,E1 25048.749,E2 25048.749} C_VEL
LIN {X 0,Y 97.825,Z 598.94,A -85,B 0,C 180,E1 25063.712,E2 25063.712} C_VEL
LIN {X 0,Y 84.738,Z 607.35,A -85,B 0,C 180,E1 25083.304,E2 25083.304} C_VEL
LIN {X 0,Y 81.482,Z 610.322,A -85,B 0,C 180,E1 25099.276,E2 25099.276} C_VEL
LIN {X 0,Y 81.765,Z 611.01,A -85,B 0,C 180,E1 25109.984,E2 25109.984} C_VEL
LIN {X 0,Y 83.245,Z 608.701,A -85,B 0,C 180,E1 25131.313,E2 25131.313} C_VEL
LIN {X 0,Y 97.389,Z 600.04,A -85,B 0,C 180,E1 25154.232,E2 25154.232} C_VEL
LIN {X 0,Y 101.928,Z 597.878,A -85,B 0,C 180,E1 25157.938,E2 25157.938} C_VEL
LIN {X 0,Y 103.252,Z 597.744,A -85,B 0,C 180,E1 25160.01,E2 25160.01} C_VEL
LIN {X 0,Y 95.99,Z 594.702,A -85,B 0,C 180,E1 25166.488,E2 25166.488} C_VEL
LIN {X 0,Y 84.352,Z 588.846,A -85,B 0,C 180,E1 25199.993,E2 25199.993} C_VEL
LIN {X 0,Y 110.316,Z 583.083,A -85,B 0,C 180,E1 25240.198,E2 25240.198} C_VEL
LIN {X 0,Y 111.172,Z 583.313,A -85,B 0,C 180,E1 25241.594,E2 25241.594} C_VEL
LIN {X 0,Y 91.407,Z 593.554,A -85,B 0,C 180,E1 25260.223,E2 25260.223} C_VEL
LIN {X 0,Y 83.453,Z 597.231,A -85,B 0,C 180,E1 25279.564,E2 25279.564} C_VEL
LIN {X 0,Y 83.455,Z 597.203,A -85,B 0,C 180,E1 25300.467,E2 25300.467} C_VEL
LIN {X 0,Y 91.459,Z 593.465,A -85,B 0,C 180,E1 25319.791,E2 25319.791} C_VEL
LIN {X 0,Y 111.362,Z 583.11,A -85,B 0,C 180,E1 25338.409,E2 25338.409} C_VEL
LIN {X 0,Y 135.782,Z 567.306,A -85,B 0,C 180,E1 25349.87,E2 25349.87} C_VEL
LIN {X 0,Y 160.427,Z 547.043,A -85,B 0,C 180,E1 25356.961,E2 25356.961} C_VEL
LIN {X 0,Y 174.736,Z 532.454,A -85,B 0,C 180,E1 25360.075,E2 25360.075} C_VEL
LIN {X 0,Y 176.733,Z 528.402,A -85,B 0,C 180,E1 25362.946,E2 25362.946} C_VEL
LIN {X 0,Y 177.335,Z 525.849,A -85,B 0,C 180,E1 25366.361,E2 25366.361} C_VEL
LIN {X 0,Y 176.218,Z 524.646,A -85,B 0,C 180,E1 25374.411,E2 25374.411} C_VEL
LIN {X 0,Y 177.237,Z 524.161,A -85,B 0,C 180,E1 25380.003,E2 25380.003} C_VEL
LIN {X 0,Y 175.379,Z 529.961,A -85,B 0,C 180,E1 25387.443,E2 25387.443} C_VEL
LIN {X 0,Y 173.98,Z 533.897,A -85,B 0,C 180,E1 25390.659,E2 25390.659} C_VEL
LIN {X 0,Y 149.239,Z 558.745,A -85,B 0,C 180,E1 25395.45,E2 25395.45} C_VEL
LIN {X 0,Y 121.752,Z 580.186,A -85,B 0,C 180,E1 25403.475,E2 25403.475} C_VEL
LIN {X 0,Y 97.902,Z 595.13,A -85,B 0,C 180,E1 25415.701,E2 25415.701} C_VEL
LIN {X 0,Y 80.01,Z 605.24,A -85,B 0,C 180,E1 25435.394,E2 25435.394} C_VEL
LIN {X 0,Y 73.656,Z 609.677,A -85,B 0,C 180,E1 25458.121,E2 25458.121} C_VEL
LIN {X 0,Y 73.858,Z 610.37,A -85,B 0,C 180,E1 25469.982,E2 25469.982} C_VEL
LIN {X 0,Y 75.8,Z 608.05,A -85,B 0,C 180,E1 25493.525,E2 25493.525} C_VEL
LIN {X 0,Y 90.753,Z 599.956,A -85,B 0,C 180,E1 25516.818,E2 25516.818} C_VEL
LIN {X 0,Y 93.947,Z 598.103,A -85,B 0,C 180,E1 25519.858,E2 25519.858} C_VEL
LIN {X 0,Y 76.904,Z 591.508,A -85,B 0,C 180,E1 25559.993,E2 25559.993} C_VEL
LIN {X 0,Y 97.849,Z 586.605,A -85,B 0,C 180,E1 25598.227,E2 25598.227} C_VEL
LIN {X 0,Y 101.1,Z 586.496,A -85,B 0,C 180,E1 25601.539,E2 25601.539} C_VEL
LIN {X 0,Y 84.621,Z 594.196,A -85,B 0,C 180,E1 25617.557,E2 25617.557} C_VEL
LIN {X 0,Y 75.723,Z 597.868,A -85,B 0,C 180,E1 25638.485,E2 25638.485} C_VEL
LIN {X 0,Y 75.729,Z 597.839,A -85,B 0,C 180,E1 25661.549,E2 25661.549} C_VEL
LIN {X 0,Y 84.679,Z 594.106,A -85,B 0,C 180,E1 25682.454,E2 25682.454} C_VEL
LIN {X 0,Y 103.695,Z 585.063,A -85,B 0,C 180,E1 25700.059,E2 25700.059} C_VEL
LIN {X 0,Y 128.902,Z 570.102,A -85,B 0,C 180,E1 25711.795,E2 25711.795} C_VEL
LIN {X 0,Y 154.195,Z 550.602,A -85,B 0,C 180,E1 25718.889,E2 25718.889} C_VEL
LIN {X 0,Y 169.717,Z 535.804,A -85,B 0,C 180,E1 25722.041,E2 25722.041} C_VEL
LIN {X 0,Y 173.44,Z 529.347,A -85,B 0,C 180,E1 25727.412,E2 25727.412} C_VEL
LIN {X 0,Y 176.218,Z 524.646,A -85,B 0,C 180,E1 25734.411,E2 25734.411} C_VEL
LIN {X 0,Y 175.77,Z 525.349,A -85,B 0,C 180,E1 25737.922,E2 25737.922} C_VEL
LIN {X 0,Y 170.257,Z 534.05,A -85,B 0,C 180,E1 25745.588,E2 25745.588} C_VEL
LIN {X 0,Y 168.543,Z 537.822,A -85,B 0,C 180,E1 25748.81,E2 25748.81} C_VEL
LIN {X 0,Y 141.825,Z 562.6,A -85,B 0,C 180,E1 25753.543,E2 25753.543} C_VEL
LIN {X 0,Y 113.936,Z 582.573,A -85,B 0,C 180,E1 25761.514,E2 25761.514} C_VEL
LIN {X 0,Y 87.598,Z 597.487,A -85,B 0,C 180,E1 25775.744,E2 25775.744} C_VEL
LIN {X 0,Y 70.898,Z 605.905,A -85,B 0,C 180,E1 25796.812,E2 25796.812} C_VEL
LIN {X 0,Y 65.837,Z 609.028,A -85,B 0,C 180,E1 25816.686,E2 25816.686} C_VEL
LIN {X 0,Y 65.927,Z 609.729,A -85,B 0,C 180,E1 25829.98,E2 25829.98} C_VEL
LIN {X 0,Y 68.492,Z 607.399,A -85,B 0,C 180,E1 25856.215,E2 25856.215} C_VEL
LIN {X 0,Y 81.911,Z 600.946,A -85,B 0,C 180,E1 25877.649,E2 25877.649} C_VEL
LIN {X 0,Y 83.632,Z 599.585,A -85,B 0,C 180,E1 25880.902,E2 25880.902} C_VEL
LIN {X 0,Y 69.368,Z 593.951,A -85,B 0,C 180,E1 25919.992,E2 25919.992} C_VEL
LIN {X 0,Y 90.826,Z 589.209,A -85,B 0,C 180,E1 25960.224,E2 25960.224} C_VEL
LIN {X 0,Y 89.705,Z 590.009,A -85,B 0,C 180,E1 25962.45,E2 25962.45} C_VEL
LIN {X 0,Y 71.932,Z 597.163,A -85,B 0,C 180,E1 25985.126,E2 25985.126} C_VEL
LIN {X 0,Y 66.815,Z 598.988,A -85,B 0,C 180,E1 26010.019,E2 26010.019} C_VEL
LIN {X 0,Y 71.998,Z 597.111,A -85,B 0,C 180,E1 26034.889,E2 26034.889} C_VEL
LIN {X 0,Y 90.385,Z 589.624,A -85,B 0,C 180,E1 26057.943,E2 26057.943} C_VEL
LIN {X 0,Y 116.06,Z 576.515,A -85,B 0,C 180,E1 26071.726,E2 26071.726} C_VEL
LIN {X 0,Y 143.172,Z 558.084,A -85,B 0,C 180,E1 26079.82,E2 26079.82} C_VEL
LIN {X 0,Y 164.725,Z 539.221,A -85,B 0,C 180,E1 26084.132,E2 26084.132} C_VEL
LIN {X 0,Y 168.765,Z 533.313,A -85,B 0,C 180,E1 26089.668,E2 26089.668} C_VEL
LIN {X 0,Y 170.976,Z 530.334,A -85,B 0,C 180,E1 26094.923,E2 26094.923} C_VEL
LIN {X 0,Y 171.837,Z 530.136,A -85,B 0,C 180,E1 26100.003,E2 26100.003} C_VEL
LIN {X 0,Y 170.257,Z 534.05,A -85,B 0,C 180,E1 26105.588,E2 26105.588} C_VEL
LIN {X 0,Y 167.011,Z 538.168,A -85,B 0,C 180,E1 26107.058,E2 26107.058} C_VEL
LIN {X 0,Y 154.112,Z 550.092,A -85,B 0,C 180,E1 26107.926,E2 26107.926} C_VEL
LIN {X 0,Y 126.437,Z 572.132,A -85,B 0,C 180,E1 26113.333,E2 26113.333} C_VEL
LIN {X 0,Y 98.395,Z 589.165,A -85,B 0,C 180,E1 26122.572,E2 26122.572} C_VEL
LIN {X 0,Y 73.588,Z 601.161,A -85,B 0,C 180,E1 26139.484,E2 26139.484} C_VEL
LIN {X 0,Y 61.219,Z 606.696,A -85,B 0,C 180,E1 26160.332,E2 26160.332} C_VEL
LIN {X 0,Y 57.992,Z 609.087,A -85,B 0,C 180,E1 26189.978,E2 26189.978} C_VEL
LIN {X 0,Y 61.384,Z 606.75,A -85,B 0,C 180,E1 26219.531,E2 26219.531} C_VEL
LIN {X 0,Y 73.992,Z 601.44,A -85,B 0,C 180,E1 26239.588,E2 26239.588} C_VEL
LIN {X 0,Y 73.594,Z 600.832,A -85,B 0,C 180,E1 26241.883,E2 26241.883} C_VEL
LIN {X 0,Y 61.766,Z 596.17,A -85,B 0,C 180,E1 26279.991,E2 26279.991} C_VEL
LIN {X 0,Y 76.638,Z 592.508,A -85,B 0,C 180,E1 26316.334,E2 26316.334} C_VEL
LIN {X 0,Y 80.789,Z 592.16,A -85,B 0,C 180,E1 26321.471,E2 26321.471} C_VEL
LIN {X 0,Y 64.838,Z 597.802,A -85,B 0,C 180,E1 26342.184,E2 26342.184} C_VEL
LIN {X 0,Y 58.949,Z 599.625,A -85,B 0,C 180,E1 26370.022,E2 26370.022} C_VEL
LIN {X 0,Y 64.907,Z 597.751,A -85,B 0,C 180,E1 26397.829,E2 26397.829} C_VEL
LIN {X 0,Y 85.288,Z 590.267,A -85,B 0,C 180,E1 26421.892,E2 26421.892} C_VEL
LIN {X 0,Y 112.522,Z 577.164,A -85,B 0,C 180,E1 26435.283,E2 26435.283} C_VEL
LIN {X 0,Y 140.652,Z 558.749,A -85,B 0,C 180,E1 26442.83,E2 26442.83} C_VEL
LIN {X 0,Y 159.76,Z 542.788,A -85,B 0,C 180,E1 26446.336,E2 26446.336} C_VEL
LIN {X 0,Y 162.524,Z 539.383,A -85,B 0,C 180,E1 26449.267,E2 26449.267} C_VEL
LIN {X 0,Y 165.259,Z 536.158,A -85,B 0,C 180,E1 26454.747,E2 26454.747} C_VEL
LIN {X 0,Y 166.191,Z 535.869,A -85,B 0,C 180,E1 26460.003,E2 26460.003} C_VEL
LIN {X 0,Y 164.157,Z 540.222,A -85,B 0,C 180,E1 26465.967,E2 26465.967} C_VEL
LIN {X 0,Y 160.69,Z 543.926,A -85,B 0,C 180,E1 26466.956,E2 26466.956} C_VEL
LIN {X 0,Y 154.112,Z 550.092,A -85,B 0,C 180,E1 26467.926,E2 26467.926} C_VEL
LIN {X 0,Y 140.333,Z 560.926,A -85,B 0,C 180,E1 26468.537,E2 26468.537} C_VEL
LIN {X 0,Y 125.969,Z 570.63,A -85,B 0,C 180,E1 26469.429,E2 26469.429} C_VEL
LIN {X 0,Y 95.55,Z 588.497,A -85,B 0,C 180,E1 26478.029,E2 26478.029} C_VEL
LIN {X 0,Y 68.694,Z 600.499,A -85,B 0,C 180,E1 26494.231,E2 26494.231} C_VEL
LIN {X 0,Y 53.842,Z 606.228,A -85,B 0,C 180,E1 26517.534,E2 26517.534} C_VEL
LIN {X 0,Y 50.05,Z 608.444,A -85,B 0,C 180,E1 26549.974,E2 26549.974} C_VEL
LIN {X 0,Y 54.545,Z 606.101,A -85,B 0,C 180,E1 26583.69,E2 26583.69} C_VEL
LIN {X 0,Y 62.004,Z 603.391,A -85,B 0,C 180,E1 26597.066,E2 26597.066} C_VEL
LIN {X 0,Y 64.18,Z 602.026,A -85,B 0,C 180,E1 26602.3,E2 26602.3} C_VEL
LIN {X 0,Y 56.645,Z 596.777,A -85,B 0,C 180,E1 26655.491,E2 26655.491} C_VEL
LIN {X 0,Y 70.573,Z 594.468,A -85,B 0,C 180,E1 26680.047,E2 26680.047} C_VEL
LIN {X 0,Y 57.972,Z 598.44,A -85,B 0,C 180,E1 26698.54,E2 26698.54} C_VEL
LIN {X 0,Y 51.072,Z 600.262,A -85,B 0,C 180,E1 26730.025,E2 26730.025} C_VEL
LIN {X 0,Y 58.043,Z 598.389,A -85,B 0,C 180,E1 26761.47,E2 26761.47} C_VEL
LIN {X 0,Y 80.858,Z 590.829,A -85,B 0,C 180,E1 26786.457,E2 26786.457} C_VEL
LIN {X 0,Y 109.451,Z 577.811,A -85,B 0,C 180,E1 26799.046,E2 26799.046} C_VEL
LIN {X 0,Y 138.522,Z 559.419,A -85,B 0,C 180,E1 26805.96,E2 26805.96} C_VEL
LIN {X 0,Y 155.737,Z 545.523,A -85,B 0,C 180,E1 26808.793,E2 26808.793} C_VEL
LIN {X 0,Y 159.225,Z 541.803,A -85,B 0,C 180,E1 26814.548,E2 26814.548} C_VEL
LIN {X 0,Y 160.336,Z 541.439,A -85,B 0,C 180,E1 26820.004,E2 26820.004} C_VEL
LIN {X 0,Y 158.971,Z 543.996,A -85,B 0,C 180,E1 26823.885,E2 26823.885} C_VEL
LIN {X 0,Y 131.957,Z 566.445,A -85,B 0,C 180,E1 26828.228,E2 26828.228} C_VEL
LIN {X 0,Y 125.969,Z 570.63,A -85,B 0,C 180,E1 26829.429,E2 26829.429} C_VEL
LIN {X 0,Y 110.99,Z 579.364,A -85,B 0,C 180,E1 26830.718,E2 26830.718} C_VEL
LIN {X 0,Y 95.462,Z 586.813,A -85,B 0,C 180,E1 26832.568,E2 26832.568} C_VEL
LIN {X 0,Y 65.006,Z 599.634,A -85,B 0,C 180,E1 26847.77,E2 26847.77} C_VEL
LIN {X 0,Y 47.813,Z 605.385,A -85,B 0,C 180,E1 26870.673,E2 26870.673} C_VEL
LIN {X 0,Y 42.12,Z 607.802,A -85,B 0,C 180,E1 26909.969,E2 26909.969} C_VEL
LIN {X 0,Y 48.049,Z 605.451,A -85,B 0,C 180,E1 26949.027,E2 26949.027} C_VEL
LIN {X 0,Y 53.655,Z 603.724,A -85,B 0,C 180,E1 26959.014,E2 26959.014} C_VEL
LIN {X 0,Y 54.591,Z 602.979,A -85,B 0,C 180,E1 26963.15,E2 26963.15} C_VEL
LIN {X 0,Y 49.259,Z 598.443,A -85,B 0,C 180,E1 27017.886,E2 27017.886} C_VEL
LIN {X 0,Y 55.964,Z 597.177,A -85,B 0,C 180,E1 27032.742,E2 27032.742} C_VEL
LIN {X 0,Y 60.23,Z 596.771,A -85,B 0,C 180,E1 27041.089,E2 27041.089} C_VEL
LIN {X 0,Y 45.306,Z 600.415,A -85,B 0,C 180,E1 27070.509,E2 27070.509} C_VEL
LIN {X 0,Y 45.325,Z 600.386,A -85,B 0,C 180,E1 27109.543,E2 27109.543} C_VEL
LIN {X 0,Y 60.418,Z 596.671,A -85,B 0,C 180,E1 27138.772,E2 27138.772} C_VEL
LIN {X 0,Y 86.823,Z 587.641,A -85,B 0,C 180,E1 27156.306,E2 27156.306} C_VEL
LIN {X 0,Y 118.511,Z 572.006,A -85,B 0,C 180,E1 27165.805,E2 27165.805} C_VEL
LIN {X 0,Y 147.165,Z 552.248,A -85,B 0,C 180,E1 27170.704,E2 27170.704} C_VEL
LIN {X 0,Y 150.086,Z 549.925,A -85,B 0,C 180,E1 27171.103,E2 27171.103} C_VEL
LIN {X 0,Y 152.422,Z 547.77,A -85,B 0,C 180,E1 27173.413,E2 27173.413} C_VEL
LIN {X 0,Y 154.291,Z 546.851,A -85,B 0,C 180,E1 27180.004,E2 27180.004} C_VEL
LIN {X 0,Y 153.77,Z 547.684,A -85,B 0,C 180,E1 27181.507,E2 27181.507} C_VEL
LIN {X 0,Y 125.523,Z 569.512,A -85,B 0,C 180,E1 27185.61,E2 27185.61} C_VEL
LIN {X 0,Y 95.462,Z 586.813,A -85,B 0,C 180,E1 27192.568,E2 27192.568} C_VEL
LIN {X 0,Y 79.627,Z 593.157,A -85,B 0,C 180,E1 27195.332,E2 27195.332} C_VEL
LIN {X 0,Y 63.743,Z 598.277,A -85,B 0,C 180,E1 27199.658,E2 27199.658} C_VEL
LIN {X 0,Y 38.368,Z 605.616,A -85,B 0,C 180,E1 27232.131,E2 27232.131} C_VEL
LIN {X 0,Y 34.167,Z 607.159,A -85,B 0,C 180,E1 27269.962,E2 27269.962} C_VEL
LIN {X 0,Y 45.001,Z 604.057,A -85,B 0,C 180,E1 27321.015,E2 27321.015} C_VEL
LIN {X 0,Y 43.068,Z 603.256,A -85,B 0,C 180,E1 27328.942,E2 27328.942} C_VEL
LIN {X 0,Y 49.524,Z 598.645,A -85,B 0,C 180,E1 27397.675,E2 27397.675} C_VEL
LIN {X 0,Y 49.482,Z 598.789,A -85,B 0,C 180,E1 27401.67,E2 27401.67} C_VEL
LIN {X 0,Y 37.98,Z 601.05,A -85,B 0,C 180,E1 27426.546,E2 27426.546} C_VEL
LIN {X 0,Y 38.003,Z 601.023,A -85,B 0,C 180,E1 27473.513,E2 27473.513} C_VEL
LIN {X 0,Y 60.284,Z 596.099,A -85,B 0,C 180,E1 27508.919,E2 27508.919} C_VEL
LIN {X 0,Y 90.814,Z 585.514,A -85,B 0,C 180,E1 27523.498,E2 27523.498} C_VEL
LIN {X 0,Y 122.789,Z 569.169,A -85,B 0,C 180,E1 27530.59,E2 27530.59} C_VEL
LIN {X 0,Y 146.457,Z 552.644,A -85,B 0,C 180,E1 27534.071,E2 27534.071} C_VEL
LIN {X 0,Y 147.757,Z 552.061,A -85,B 0,C 180,E1 27538.639,E2 27538.639} C_VEL
LIN {X 0,Y 147.041,Z 552.746,A -85,B 0,C 180,E1 27539.36,E2 27539.36} C_VEL
LIN {X 0,Y 116.265,Z 574.277,A -85,B 0,C 180,E1 27543.227,E2 27543.227} C_VEL
LIN {X 0,Y 85.193,Z 590.168,A -85,B 0,C 180,E1 27550.243,E2 27550.243} C_VEL
LIN {X 0,Y 63.743,Z 598.277,A -85,B 0,C 180,E1 27559.658,E2 27559.658} C_VEL
LIN {X 0,Y 56.228,Z 600.44,A -85,B 0,C 180,E1 27563.464,E2 27563.464} C_VEL
LIN {X 0,Y 34.963,Z 604.431,A -85,B 0,C 180,E1 27577.781,E2 27577.781} C_VEL
LIN {X 0,Y 33.519,Z 604.618,A -85,B 0,C 180,E1 27580.534,E2 27580.534} C_VEL
LIN {X 0,Y 26.208,Z 606.515,A -85,B 0,C 180,E1 27629.951,E2 27629.951} C_VEL
LIN {X 0,Y 34.878,Z 604.55,A -85,B 0,C 180,E1 27681.224,E2 27681.224} C_VEL
LIN {X 0,Y 34.841,Z 604.044,A -85,B 0,C 180,E1 27687.529,E2 27687.529} C_VEL
LIN {X 0,Y 34.754,Z 601.095,A -85,B 0,C 180,E1 27745.806,E2 27745.806} C_VEL
LIN {X 0,Y 39.729,Z 600.355,A -85,B 0,C 180,E1 27760.398,E2 27760.398} C_VEL
LIN {X 0,Y 27.465,Z 602.172,A -85,B 0,C 180,E1 27810.047,E2 27810.047} C_VEL
LIN {X 0,Y 39.798,Z 600.307,A -85,B 0,C 180,E1 27859.585,E2 27859.585} C_VEL
LIN {X 0,Y 67.821,Z 593.642,A -85,B 0,C 180,E1 27881.63,E2 27881.63} C_VEL
LIN {X 0,Y 98.699,Z 581.912,A -85,B 0,C 180,E1 27890.533,E2 27890.533} C_VEL
LIN {X 0,Y 131.026,Z 563.99,A -85,B 0,C 180,E1 27895.375,E2 27895.375} C_VEL
LIN {X 0,Y 140.833,Z 557.152,A -85,B 0,C 180,E1 27896.635,E2 27896.635} C_VEL
LIN {X 0,Y 108.011,Z 578.128,A -85,B 0,C 180,E1 27900.295,E2 27900.295} C_VEL
LIN {X 0,Y 76.271,Z 592.568,A -85,B 0,C 180,E1 27906.898,E2 27906.898} C_VEL
LIN {X 0,Y 48.544,Z 601.284,A -85,B 0,C 180,E1 27920.598,E2 27920.598} C_VEL
LIN {X 0,Y 33.519,Z 604.618,A -85,B 0,C 180,E1 27940.534,E2 27940.534} C_VEL
LIN {X 0,Y 25,Z 605.789,A -85,B 0,C 180,E1 27960.253,E2 27960.253} C_VEL
LIN {X 0,Y 19.351,Z 605.429,A -85,B 0,C 180,E1 28019.301,E2 28019.301} C_VEL
LIN {X 0,Y 25.213,Z 604.748,A -85,B 0,C 180,E1 28043.07,E2 28043.07} C_VEL
LIN {X 0,Y 22.905,Z 603.275,A -85,B 0,C 180,E1 28079.975,E2 28079.975} C_VEL
LIN {X 0,Y 27.873,Z 601.992,A -85,B 0,C 180,E1 28112.874,E2 28112.874} C_VEL
LIN {X 0,Y 28.295,Z 601.937,A -85,B 0,C 180,E1 28121.056,E2 28121.056} C_VEL
LIN {X 0,Y 19.588,Z 602.81,A -85,B 0,C 180,E1 28170.066,E2 28170.066} C_VEL
LIN {X 0,Y 35.197,Z 600.945,A -85,B 0,C 180,E1 28229.418,E2 28229.418} C_VEL
LIN {X 0,Y 65.753,Z 594.288,A -85,B 0,C 180,E1 28248.205,E2 28248.205} C_VEL
LIN {X 0,Y 99.323,Z 581.829,A -85,B 0,C 180,E1 28255.358,E2 28255.358} C_VEL
LIN {X 0,Y 104.188,Z 579.593,A -85,B 0,C 180,E1 28256.042,E2 28256.042} C_VEL
LIN {X 0,Y 71.962,Z 593.241,A -85,B 0,C 180,E1 28261.6,E2 28261.6} C_VEL
LIN {X 0,Y 39.396,Z 602.131,A -85,B 0,C 180,E1 28275.997,E2 28275.997} C_VEL
LIN {X 0,Y 21.954,Z 605.128,A -85,B 0,C 180,E1 28306.322,E2 28306.322} C_VEL
LIN {X 0,Y 18.242,Z 605.87,A -85,B 0,C 180,E1 28349.929,E2 28349.929} C_VEL
LIN {X 0,Y 19.351,Z 605.429,A -85,B 0,C 180,E1 28379.301,E2 28379.301} C_VEL
LIN {X 0,Y 17.99,Z 605.035,A -85,B 0,C 180,E1 28395.806,E2 28395.806} C_VEL
LIN {X 0,Y 14.995,Z 604.413,A -85,B 0,C 180,E1 28417.753,E2 28417.753} C_VEL
LIN {X 0,Y 18.809,Z 602.963,A -85,B 0,C 180,E1 28476.516,E2 28476.516} C_VEL
LIN {X 0,Y 18.853,Z 602.936,A -85,B 0,C 180,E1 28583.534,E2 28583.534} C_VEL
LIN {X 0,Y 46.172,Z 599.235,A -85,B 0,C 180,E1 28609.79,E2 28609.79} C_VEL
LIN {X 0,Y 66.242,Z 594.482,A -85,B 0,C 180,E1 28615.994,E2 28615.994} C_VEL
LIN {X 0,Y 30.641,Z 602.761,A -85,B 0,C 180,E1 28628.542,E2 28628.542} C_VEL
LIN {X 0,Y 10.283,Z 605.226,A -85,B 0,C 180,E1 28709.874,E2 28709.874} C_VEL
LIN {X 0,Y 15.511,Z 604.59,A -85,B 0,C 180,E1 28770.747,E2 28770.747} C_VEL
LIN {X 0,Y 14.995,Z 604.413,A -85,B 0,C 180,E1 28777.753,E2 28777.753} C_VEL
LIN {X 0,Y 11.16,Z 604.175,A -85,B 0,C 180,E1 28797.531,E2 28797.531} C_VEL
LIN {X 0,Y 4.16,Z 604.122,A -85,B 0,C 180,E1 28842.327,E2 28842.327} C_VEL
LIN {X 0,Y 8.462,Z 603.825,A -85,B 0,C 180,E1 28954.872,E2 28954.872} C_VEL
LIN {X 0,Y 22.387,Z 603.161,A -85,B 0,C 180,E1 28975.448,E2 28975.448} C_VEL
LIN {X 0,Y 2.303,Z 604.581,A -85,B 0,C 180,E1 29069.438,E2 29069.438} C_VEL
LIN {X 0,Y 6.876,Z 604.251,A -85,B 0,C 180,E1 29159.917,E2 29159.917} C_VEL
LIN {X 0,Y 7.423,Z 604.088,A -85,B 0,C 180,E1 29174.953,E2 29174.953} C_VEL
LIN {X 0,Y 3.856,Z 604.083,A -85,B 0,C 180,E1 29250.336,E2 29250.336} C_VEL
LIN {X 0,Y 8.462,Z 603.825,A -85,B 0,C 180,E1 29314.872,E2 29314.872} C_VEL
LIN {X 0,Y 10.345,Z 605.824,A -85,B 0,C 180,E1 29320.094,E2 29320.094} C_VEL
LIN {X 0,Y 10.345,Z 647,A -85,B 0,C 180,E1 29320.094,E2 29320.094} C_VEL
LIN {X 0,Y 10.345,Z 647,A -85,B 0,C 180,E1 29320.094,E2 29320.094}

QRS_NEXT_CUT()
PTP {E1 29336.932,E2 29336.932}
PTP {X 0,Y 607.864,A -85,B 0,C 180,E1 29336.932,E2 29336.932,E3 0,E4 0,E5 0,E6 0}
QRS_SPEED_INIT()
LIN {X 0,Y 607.864,Z 647,A -85,B 0,C 180,E1 29336.932,E2 29336.932,E3 0,E4 0,E5 0,E6 0} C_VEL
LIN {X 0,Y 607.864,Z 103.84,A -85,B 0,C 180,E1 29336.932,E2 29336.932} C_VEL
LIN {X 0,Y 607.864,Z 95.763,A -85,B 0,C 180,E1 29336.932,E2 29336.932} C_VEL
LIN {X 0,Y 607.886,Z 93.763,A -85,B 0,C 180,E1 29336.743,E2 29336.743} C_VEL
LIN {X 0,Y 607.842,Z 93.764,A -85,B 0,C 180,E1 29333.672,E2 29333.672} C_VEL
LIN {X 0,Y 607.893,Z 93.763,A -85,B 0,C 180,E1 29330.724,E2 29330.724} C_VEL
LIN {X 0,Y 607.839,Z 93.764,A -85,B 0,C 180,E1 29327.652,E2 29327.652} C_VEL
LIN {X 0,Y 607.905,Z 93.764,A -85,B 0,C 180,E1 29324.644,E2 29324.644} C_VEL
LIN {X 0,Y 607.836,Z 93.764,A -85,B 0,C 180,E1 29321.644,E2 29321.644} C_VEL
LIN {X 0,Y 607.91,Z 93.766,A -85,B 0,C 180,E1 29318.577,E2 29318.577} C_VEL
LIN {X 0,Y 607.833,Z 93.764,A -85,B 0,C 180,E1 29315.614,E2 29315.614} C_VEL
LIN {X 0,Y 607.915,Z 93.764,A -85,B 0,C 180,E1 29312.579,E2 29312.579} C_VEL
LIN {X 0,Y 607.834,Z 93.764,A -85,B 0,C 180,E1 29309.535,E2 29309.535} C_VEL
LIN {X 0,Y 607.887,Z 93.765,A -85,B 0,C 180,E1 29306.45,E2 29306.45} C_VEL
LIN {X 0,Y 607.833,Z 93.765,A -85,B 0,C 180,E1 29303.549,E2 29303.549} C_VEL
LIN {X 0,Y 607.882,Z 93.765,A -85,B 0,C 180,E1 29300.465,E2 29300.465} C_VEL
LIN {X 0,Y 607.831,Z 93.765,A -85,B 0,C 180,E1 29297.589,E2 29297.589} C_VEL
LIN {X 0,Y 607.877,Z 93.765,A -85,B 0,C 180,E1 29294.482,E2 29294.482} C_VEL
LIN {X 0,Y 607.831,Z 93.765,A -85,B 0,C 180,E1 29291.648,E2 29291.648} C_VEL
LIN {X 0,Y 607.884,Z 93.765,A -85,B 0,C 180,E1 29288.563,E2 29288.563} C_VEL
LIN {X 0,Y 607.833,Z 93.765,A -85,B 0,C 180,E1 29285.648,E2 29285.648} C_VEL
LIN {X 0,Y 607.876,Z 93.765,A -85,B 0,C 180,E1 29282.537,E2 29282.537} C_VEL
LIN {X 0,Y 607.835,Z 93.765,A -85,B 0,C 180,E1 29279.677,E2 29279.677} C_VEL
LIN {X 0,Y 607.853,Z 93.888,A -85,B 0,C 180,E1 29278.335,E2 29278.335} C_VEL
LIN {X 0,Y 607.87,Z 131.132,A -85,B 0,C 180,E1 29275.527,E2 29275.527} C_VEL
LIN {X 0,Y 607.882,Z 173.343,A -85,B 0,C 180,E1 29272.423,E2 29272.423} C_VEL
LIN {X 0,Y 607.878,Z 175.714,A -85,B 0,C 180,E1 29272.273,E2 29272.273} C_VEL
LIN {X 0,Y 607.914,Z 383.967,A -85,B 0,C 180,E1 29269.666,E2 29269.666} C_VEL
LIN {X 0,Y 607.915,Z 402.888,A -85,B 0,C 180,E1 29269.251,E2 29269.251} C_VEL
LIN {X 0,Y 607.916,Z 421.151,A -85,B 0,C 180,E1 29268.672,E2 29268.672} C_VEL
LIN {X 0,Y 607.916,Z 439.166,A -85,B 0,C 180,E1 29267.912,E2 29267.912} C_VEL
LIN {X 0,Y 607.919,Z 455.873,A -85,B 0,C 180,E1 29267.023,E2 29267.023} C_VEL
LIN {X 0,Y 607.918,Z 471.707,A -85,B 0,C 180,E1 29265.991,E2 29265.991} C_VEL
LIN {X 0,Y 607.915,Z 486.614,A -85,B 0,C 180,E1 29264.818,E2 29264.818} C_VEL
LIN {X 0,Y 607.916,Z 500.523,A -85,B 0,C 180,E1 29263.506,E2 29263.506} C_VEL
LIN {X 0,Y 607.916,Z 513.326,A -85,B 0,C 180,E1 29262.056,E2 29262.056} C_VEL
LIN {X 0,Y 607.911,Z 524.568,A -85,B 0,C 180,E1 29260.519,E2 29260.519} C_VEL
LIN {X 0,Y 607.915,Z 534.266,A -85,B 0,C 180,E1 29258.893,E2 29258.893} C_VEL
LIN {X 0,Y 607.909,Z 541.989,A -85,B 0,C 180,E1 29257.275,E2 29257.275} C_VEL
LIN {X 0,Y 607.91,Z 548.268,A -85,B 0,C 180,E1 29255.568,E2 29255.568} C_VEL
LIN {X 0,Y 607.917,Z 552.981,A -85,B 0,C 180,E1 29253.772,E2 29253.772} C_VEL
LIN {X 0,Y 607.918,Z 555.846,A -85,B 0,C 180,E1 29251.979,E2 29251.979} C_VEL
LIN {X 0,Y 607.91,Z 556.951,A -85,B 0,C 180,E1 29250.188,E2 29250.188} C_VEL
LIN {X 0,Y 607.915,Z 556.313,A -85,B 0,C 180,E1 29248.397,E2 29248.397} C_VEL
LIN {X 0,Y 607.907,Z 553.922,A -85,B 0,C 180,E1 29246.605,E2 29246.605} C_VEL
LIN {X 0,Y 607.911,Z 549.709,A -85,B 0,C 180,E1 29244.809,E2 29244.809} C_VEL
LIN {X 0,Y 607.919,Z 543.927,A -85,B 0,C 180,E1 29243.104,E2 29243.104} C_VEL
LIN {X 0,Y 607.91,Z 536.716,A -85,B 0,C 180,E1 29241.487,E2 29241.487} C_VEL
LIN {X 0,Y 607.917,Z 527.623,A -85,B 0,C 180,E1 29239.863,E2 29239.863} C_VEL
LIN {X 0,Y 607.914,Z 517.06,A -85,B 0,C 180,E1 29238.328,E2 29238.328} C_VEL
LIN {X 0,Y 607.918,Z 504.548,A -85,B 0,C 180,E1 29236.826,E2 29236.826} C_VEL
LIN {X 0,Y 607.914,Z 490.931,A -85,B 0,C 180,E1 29235.473,E2 29235.473} C_VEL
LIN {X 0,Y 607.918,Z 476.208,A -85,B 0,C 180,E1 29234.253,E2 29234.253} C_VEL
LIN {X 0,Y 607.918,Z 460.534,A -85,B 0,C 180,E1 29233.173,E2 29233.173} C_VEL
LIN {X 0,Y 607.915,Z 443.888,A -85,B 0,C 180,E1 29232.233,E2 29232.233} C_VEL
LIN {X 0,Y 607.915,Z 426.383,A -85,B 0,C 180,E1 29231.442,E2 29231.442} C_VEL
LIN {X 0,Y 607.917,Z 408.459,A -85,B 0,C 180,E1 29230.82,E2 29230.82} C_VEL
LIN {X 0,Y 607.911,Z 390.525,A -85,B 0,C 180,E1 29230.37,E2 29230.37} C_VEL
LIN {X 0,Y 607.909,Z 370.665,A -85,B 0,C 180,E1 29230.057,E2 29230.057} C_VEL
LIN {X 0,Y 607.885,Z 175.202,A -85,B 0,C 180,E1 29227.623,E2 29227.623} C_VEL
LIN {X 0,Y 607.885,Z 132.882,A -85,B 0,C 180,E1 29224.514,E2 29224.514} C_VEL
LIN {X 0,Y 607.853,Z 95.825,A -85,B 0,C 180,E1 29221.723,E2 29221.723} C_VEL
LIN {X 0,Y 607.866,Z 93.767,A -85,B 0,C 180,E1 29221.563,E2 29221.563} C_VEL
LIN {X 0,Y 607.843,Z 93.765,A -85,B 0,C 180,E1 29218.438,E2 29218.438} C_VEL
LIN {X 0,Y 607.911,Z 93.766,A -85,B 0,C 180,E1 29215.428,E2 29215.428} C_VEL
LIN {X 0,Y 607.862,Z 93.763,A -85,B 0,C 180,E1 29212.273,E2 29212.273} C_VEL
LIN {X 0,Y 607.906,Z 93.758,A -85,B 0,C 180,E1 29209.109,E2 29209.109} C_VEL
LIN {X 0,Y 607.914,Z 93.765,A -85,B 0,C 180,E1 29205.915,E2 29205.915} C_VEL
LIN {X 0,Y 607.89,Z 93.759,A -85,B 0,C 180,E1 29202.79,E2 29202.79} C_VEL
LIN {X 0,Y 607.901,Z 93.759,A -85,B 0,C 180,E1 29199.656,E2 29199.656} C_VEL
LIN {X 0,Y 607.918,Z 93.765,A -85,B 0,C 180,E1 29196.424,E2 29196.424} C_VEL
LIN {X 0,Y 607.912,Z 93.757,A -85,B 0,C 180,E1 29193.157,E2 29193.157} C_VEL
LIN {X 0,Y 607.876,Z 93.761,A -85,B 0,C 180,E1 29190.002,E2 29190.002} C_VEL
LIN {X 0,Y 607.877,Z 93.833,A -85,B 0,C 180,E1 29188.338,E2 29188.338} C_VEL
LIN {X 0,Y 607.919,Z 133.923,A -85,B 0,C 180,E1 29185.317,E2 29185.317} C_VEL
LIN {X 0,Y 607.847,Z 174.603,A -85,B 0,C 180,E1 29182.332,E2 29182.332} C_VEL
LIN {X 0,Y 607.849,Z 176.141,A -85,B 0,C 180,E1 29182.269,E2 29182.269} C_VEL
LIN {X 0,Y 607.916,Z 383.907,A -85,B 0,C 180,E1 29179.667,E2 29179.667} C_VEL
LIN {X 0,Y 607.919,Z 402.832,A -85,B 0,C 180,E1 29179.252,E2 29179.252} C_VEL
LIN {X 0,Y 607.913,Z 421.176,A -85,B 0,C 180,E1 29178.671,E2 29178.671} C_VEL
LIN {X 0,Y 607.916,Z 439.16,A -85,B 0,C 180,E1 29177.913,E2 29177.913} C_VEL
LIN {X 0,Y 607.92,Z 456.665,A -85,B 0,C 180,E1 29176.974,E2 29176.974} C_VEL
LIN {X 0,Y 607.917,Z 472.356,A -85,B 0,C 180,E1 29175.943,E2 29175.943} C_VEL
LIN {X 0,Y 607.915,Z 487.541,A -85,B 0,C 180,E1 29174.736,E2 29174.736} C_VEL
LIN {X 0,Y 607.913,Z 501.445,A -85,B 0,C 180,E1 29173.41,E2 29173.41} C_VEL
LIN {X 0,Y 607.915,Z 514.089,A -85,B 0,C 180,E1 29171.961,E2 29171.961} C_VEL
LIN {X 0,Y 607.92,Z 525.204,A -85,B 0,C 180,E1 29170.424,E2 29170.424} C_VEL
LIN {X 0,Y 607.915,Z 534.777,A -85,B 0,C 180,E1 29168.799,E2 29168.799} C_VEL
LIN {X 0,Y 607.907,Z 542.393,A -85,B 0,C 180,E1 29167.181,E2 29167.181} C_VEL
LIN {X 0,Y 607.917,Z 548.567,A -85,B 0,C 180,E1 29165.474,E2 29165.474} C_VEL
LIN {X 0,Y 607.917,Z 552.98,A -85,B 0,C 180,E1 29163.772,E2 29163.772} C_VEL
LIN {X 0,Y 607.907,Z 555.845,A -85,B 0,C 180,E1 29161.98,E2 29161.98} C_VEL
LIN {X 0,Y 607.913,Z 556.952,A -85,B 0,C 180,E1 29160.189,E2 29160.189} C_VEL
LIN {X 0,Y 607.915,Z 556.314,A -85,B 0,C 180,E1 29158.398,E2 29158.398} C_VEL
LIN {X 0,Y 607.917,Z 553.922,A -85,B 0,C 180,E1 29156.606,E2 29156.606} C_VEL
LIN {X 0,Y 607.904,Z 549.965,A -85,B 0,C 180,E1 29154.905,E2 29154.905} C_VEL
LIN {X 0,Y 607.914,Z 544.281,A -85,B 0,C 180,E1 29153.199,E2 29153.199} C_VEL
LIN {X 0,Y 607.914,Z 537.182,A -85,B 0,C 180,E1 29151.583,E2 29151.583} C_VEL
LIN {X 0,Y 607.91,Z 528.202,A -85,B 0,C 180,E1 29149.96,E2 29149.96} C_VEL
LIN {X 0,Y 607.916,Z 517.773,A -85,B 0,C 180,E1 29148.425,E2 29148.425} C_VEL
LIN {X 0,Y 607.914,Z 505.893,A -85,B 0,C 180,E1 29146.978,E2 29146.978} C_VEL
LIN {X 0,Y 607.92,Z 492.032,A -85,B 0,C 180,E1 29145.571,E2 29145.571} C_VEL
LIN {X 0,Y 607.918,Z 476.883,A -85,B 0,C 180,E1 29144.303,E2 29144.303} C_VEL
LIN {X 0,Y 607.919,Z 461.419,A -85,B 0,C 180,E1 29143.228,E2 29143.228} C_VEL
LIN {X 0,Y 607.912,Z 444.956,A -85,B 0,C 180,E1 29142.285,E2 29142.285} C_VEL
LIN {X 0,Y 607.918,Z 427.675,A -85,B 0,C 180,E1 29141.493,E2 29141.493} C_VEL
LIN {X 0,Y 607.915,Z 410.227,A -85,B 0,C 180,E1 29140.87,E2 29140.87} C_VEL
LIN {X 0,Y 607.911,Z 391.868,A -85,B 0,C 180,E1 29140.396,E2 29140.396} C_VEL
LIN {X 0,Y 607.914,Z 372.758,A -85,B 0,C 180,E1 29140.083,E2 29140.083} C_VEL
LIN {X 0,Y 607.912,Z 175.157,A -85,B 0,C 180,E1 29137.62,E2 29137.62} C_VEL
LIN {X 0,Y 607.896,Z 132.333,A -85,B 0,C 180,E1 29134.473,E2 29134.473} C_VEL
LIN {X 0,Y 607.916,Z 93.76,A -85,B 0,C 180,E1 29131.566,E2 29131.566} C_VEL
LIN {X 0,Y 607.871,Z 93.761,A -85,B 0,C 180,E1 29128.434,E2 29128.434} C_VEL
LIN {X 0,Y 607.912,Z 93.765,A -85,B 0,C 180,E1 29125.314,E2 29125.314} C_VEL
LIN {X 0,Y 607.864,Z 93.761,A -85,B 0,C 180,E1 29122.274,E2 29122.274} C_VEL
LIN {X 0,Y 607.863,Z 93.764,A -85,B 0,C 180,E1 29118.982,E2 29118.982} C_VEL
LIN {X 0,Y 607.889,Z 93.763,A -85,B 0,C 180,E1 29115.954,E2 29115.954} C_VEL
LIN {X 0,Y 607.839,Z 93.765,A -85,B 0,C 180,E1 29112.923,E2 29112.923} C_VEL
LIN {X 0,Y 607.901,Z 93.765,A -85,B 0,C 180,E1 29109.901,E2 29109.901} C_VEL
LIN {X 0,Y 607.841,Z 93.764,A -85,B 0,C 180,E1 29106.899,E2 29106.899} C_VEL
LIN {X 0,Y 607.914,Z 93.763,A -85,B 0,C 180,E1 29103.841,E2 29103.841} C_VEL
LIN {X 0,Y 607.911,Z 93.952,A -85,B 0,C 180,E1 29101.841,E2 29101.841} C_VEL
LIN {X 0,Y 607.91,Z 144.851,A -85,B 0,C 180,E1 29098.759,E2 29098.759} C_VEL
LIN {X 0,Y 607.918,Z 163.106,A -85,B 0,C 180,E1 29097.687,E2 29097.687} C_VEL
LIN {X 0,Y 607.905,Z 402.311,A -85,B 0,C 180,E1 29094.604,E2 29094.604} C_VEL
LIN {X 0,Y 607.919,Z 428.302,A -85,B 0,C 180,E1 29094.228,E2 29094.228} C_VEL
LIN {X 0,Y 607.917,Z 447.725,A -85,B 0,C 180,E1 29093.79,E2 29093.79} C_VEL
LIN {X 0,Y 607.913,Z 467.596,A -85,B 0,C 180,E1 29093.16,E2 29093.16} C_VEL
LIN {X 0,Y 607.907,Z 486.739,A -85,B 0,C 180,E1 29092.38,E2 29092.38} C_VEL
LIN {X 0,Y 607.918,Z 505.824,A -85,B 0,C 180,E1 29091.416,E2 29091.416} C_VEL
LIN {X 0,Y 607.917,Z 523.141,A -85,B 0,C 180,E1 29090.365,E2 29090.365} C_VEL
LIN {X 0,Y 607.914,Z 540.559,A -85,B 0,C 180,E1 29089.106,E2 29089.106} C_VEL
LIN {X 0,Y 607.916,Z 557.359,A -85,B 0,C 180,E1 29087.666,E2 29087.666} C_VEL
LIN {X 0,Y 607.909,Z 572.444,A -85,B 0,C 180,E1 29086.139,E2 29086.139} C_VEL
LIN {X 0,Y 607.914,Z 585.582,A -85,B 0,C 180,E1 29084.575,E2 29084.575} C_VEL
LIN {X 0,Y 607.918,Z 597.37,A -85,B 0,C 180,E1 29082.926,E2 29082.926} C_VEL
LIN {X 0,Y 607.917,Z 608.32,A -85,B 0,C 180,E1 29081.095,E2 29081.095} C_VEL
LIN {X 0,Y 607.913,Z 617.245,A -85,B 0,C 180,E1 29079.276,E2 29079.276} C_VEL
LIN {X 0,Y 607.911,Z 624.377,A -85,B 0,C 180,E1 29077.466,E2 29077.466} C_VEL
LIN {X 0,Y 607.91,Z 630,A -85,B 0,C 180,E1 29075.569,E2 29075.569} C_VEL
LIN {X 0,Y 607.91,Z 633.923,A -85,B 0,C 180,E1 29073.678,E2 29073.678} C_VEL
LIN {X 0,Y 607.906,Z 636.305,A -85,B 0,C 180,E1 29071.697,E2 29071.697} C_VEL
LIN {X 0,Y 607.907,Z 636.962,A -85,B 0,C 180,E1 29069.812,E2 29069.812} C_VEL
LIN {X 0,Y 607.91,Z 636.04,A -85,B 0,C 180,E1 29067.927,E2 29067.927} C_VEL
LIN {X 0,Y 607.917,Z 633.451,A -85,B 0,C 180,E1 29066.04,E2 29066.04} C_VEL
LIN {X 0,Y 607.912,Z 629.243,A -85,B 0,C 180,E1 29064.148,E2 29064.148} C_VEL
LIN {X 0,Y 607.916,Z 623.329,A -85,B 0,C 180,E1 29062.25,E2 29062.25} C_VEL
LIN {X 0,Y 607.911,Z 616.019,A -85,B 0,C 180,E1 29060.438,E2 29060.438} C_VEL
LIN {X 0,Y 607.909,Z 606.675,A -85,B 0,C 180,E1 29058.599,E2 29058.599} C_VEL
LIN {X 0,Y 607.91,Z 596.099,A -85,B 0,C 180,E1 29056.882,E2 29056.882} C_VEL
LIN {X 0,Y 607.915,Z 584.041,A -85,B 0,C 180,E1 29055.231,E2 29055.231} C_VEL
LIN {X 0,Y 607.911,Z 570.602,A -85,B 0,C 180,E1 29053.666,E2 29053.666} C_VEL
LIN {X 0,Y 607.916,Z 555.716,A -85,B 0,C 180,E1 29052.187,E2 29052.187} C_VEL
LIN {X 0,Y 607.914,Z 539.917,A -85,B 0,C 180,E1 29050.846,E2 29050.846} C_VEL
LIN {X 0,Y 607.916,Z 522.544,A -85,B 0,C 180,E1 29049.594,E2 29049.594} C_VEL
LIN {X 0,Y 607.919,Z 504.066,A -85,B 0,C 180,E1 29048.484,E2 29048.484} C_VEL
LIN {X 0,Y 607.909,Z 485.621,A -85,B 0,C 180,E1 29047.569,E2 29047.569} C_VEL
LIN {X 0,Y 607.913,Z 466.328,A -85,B 0,C 180,E1 29046.795,E2 29046.795} C_VEL
LIN {X 0,Y 607.917,Z 446.741,A -85,B 0,C 180,E1 29046.186,E2 29046.186} C_VEL
LIN {X 0,Y 607.918,Z 427.072,A -85,B 0,C 180,E1 29045.748,E2 29045.748} C_VEL
LIN {X 0,Y 607.906,Z 390.003,A -85,B 0,C 180,E1 29045.24,E2 29045.24} C_VEL
LIN {X 0,Y 607.918,Z 162.721,A -85,B 0,C 180,E1 29042.301,E2 29042.301} C_VEL
LIN {X 0,Y 607.861,Z 112.458,A -85,B 0,C 180,E1 29039.288,E2 29039.288} C_VEL
LIN {X 0,Y 607.913,Z 93.763,A -85,B 0,C 180,E1 29038.133,E2 29038.133} C_VEL
LIN {X 0,Y 607.854,Z 93.763,A -85,B 0,C 180,E1 29035.081,E2 29035.081} C_VEL
LIN {X 0,Y 607.916,Z 93.764,A -85,B 0,C 180,E1 29031.983,E2 29031.983} C_VEL
LIN {X 0,Y 607.853,Z 93.762,A -85,B 0,C 180,E1 29028.982,E2 29028.982} C_VEL
LIN {X 0,Y 607.893,Z 93.764,A -85,B 0,C 180,E1 29025.783,E2 29025.783} C_VEL
LIN {X 0,Y 607.86,Z 93.761,A -85,B 0,C 180,E1 29022.792,E2 29022.792} C_VEL
LIN {X 0,Y 607.862,Z 93.762,A -85,B 0,C 180,E1 29019.517,E2 29019.517} C_VEL
LIN {X 0,Y 607.886,Z 93.76,A -85,B 0,C 180,E1 29016.543,E2 29016.543} C_VEL
LIN {X 0,Y 607.854,Z 93.763,A -85,B 0,C 180,E1 29013.438,E2 29013.438} C_VEL
LIN {X 0,Y 607.904,Z 93.761,A -85,B 0,C 180,E1 29010.437,E2 29010.437} C_VEL
LIN {X 0,Y 607.848,Z 93.763,A -85,B 0,C 180,E1 29007.347,E2 29007.347} C_VEL
LIN {X 0,Y 607.915,Z 93.763,A -85,B 0,C 180,E1 29004.279,E2 29004.279} C_VEL
LIN {X 0,Y 607.845,Z 93.763,A -85,B 0,C 180,E1 29001.216,E2 29001.216} C_VEL
LIN {X 0,Y 607.902,Z 93.765,A -85,B 0,C 180,E1 28998.111,E2 28998.111} C_VEL
LIN {X 0,Y 607.847,Z 93.763,A -85,B 0,C 180,E1 28995.161,E2 28995.161} C_VEL
LIN {X 0,Y 607.889,Z 93.764,A -85,B 0,C 180,E1 28992.057,E2 28992.057} C_VEL
LIN {X 0,Y 607.846,Z 93.763,A -85,B 0,C 180,E1 28989.181,E2 28989.181} C_VEL
LIN {X 0,Y 607.881,Z 93.764,A -85,B 0,C 180,E1 28986.042,E2 28986.042} C_VEL
LIN {X 0,Y 607.846,Z 93.763,A -85,B 0,C 180,E1 28983.189,E2 28983.189} C_VEL
LIN {X 0,Y 607.87,Z 93.764,A -85,B 0,C 180,E1 28980,E2 28980} C_VEL
LIN {X 0,Y 607.847,Z 93.763,A -85,B 0,C 180,E1 28977.171,E2 28977.171} C_VEL
LIN {X 0,Y 607.886,Z 93.763,A -85,B 0,C 180,E1 28976.743,E2 28976.743} C_VEL
LIN {X 0,Y 606.95,Z 93.886,A -85,B 0,C 180,E1 28976.017,E2 28976.017} C_VEL
LIN {X 0,Y 600.443,Z 94.69,A -85,B 0,C 180,E1 28973.98,E2 28973.98} C_VEL
LIN {X 0,Y 599.9,Z 94.752,A -85,B 0,C 180,E1 28973.45,E2 28973.45} C_VEL
LIN {X 0,Y 599.97,Z 94.754,A -85,B 0,C 180,E1 28970.407,E2 28970.407} C_VEL
LIN {X 0,Y 599.901,Z 94.752,A -85,B 0,C 180,E1 28967.388,E2 28967.388} C_VEL
LIN {X 0,Y 599.939,Z 94.753,A -85,B 0,C 180,E1 28964.237,E2 28964.237} C_VEL
LIN {X 0,Y 599.902,Z 94.752,A -85,B 0,C 180,E1 28961.336,E2 28961.336} C_VEL
LIN {X 0,Y 599.927,Z 94.753,A -85,B 0,C 180,E1 28958.171,E2 28958.171} C_VEL
LIN {X 0,Y 599.904,Z 94.753,A -85,B 0,C 180,E1 28955.27,E2 28955.27} C_VEL
LIN {X 0,Y 599.904,Z 94.752,A -85,B 0,C 180,E1 28951.965,E2 28951.965} C_VEL
LIN {X 0,Y 599.92,Z 94.753,A -85,B 0,C 180,E1 28949.114,E2 28949.114} C_VEL
LIN {X 0,Y 599.899,Z 94.754,A -85,B 0,C 180,E1 28945.929,E2 28945.929} C_VEL
LIN {X 0,Y 599.935,Z 94.753,A -85,B 0,C 180,E1 28943.012,E2 28943.012} C_VEL
LIN {X 0,Y 599.895,Z 94.754,A -85,B 0,C 180,E1 28939.908,E2 28939.908} C_VEL
LIN {X 0,Y 599.956,Z 94.754,A -85,B 0,C 180,E1 28936.881,E2 28936.881} C_VEL
LIN {X 0,Y 599.89,Z 94.754,A -85,B 0,C 180,E1 28933.805,E2 28933.805} C_VEL
LIN {X 0,Y 599.968,Z 94.755,A -85,B 0,C 180,E1 28930.788,E2 28930.788} C_VEL
LIN {X 0,Y 599.892,Z 94.754,A -85,B 0,C 180,E1 28927.811,E2 28927.811} C_VEL
LIN {X 0,Y 599.963,Z 94.755,A -85,B 0,C 180,E1 28924.746,E2 28924.746} C_VEL
LIN {X 0,Y 599.894,Z 94.755,A -85,B 0,C 180,E1 28921.781,E2 28921.781} C_VEL
LIN {X 0,Y 599.964,Z 94.848,A -85,B 0,C 180,E1 28918.668,E2 28918.668} C_VEL
LIN {X 0,Y 600.461,Z 98.179,A -85,B 0,C 180,E1 28918.385,E2 28918.385} C_VEL
LIN {X 0,Y 600.401,Z 136.055,A -85,B 0,C 180,E1 28915.497,E2 28915.497} C_VEL
LIN {X 0,Y 600.329,Z 175.662,A -85,B 0,C 180,E1 28912.57,E2 28912.57} C_VEL
LIN {X 0,Y 600.384,Z 351.287,A -85,B 0,C 180,E1 28910.355,E2 28910.355} C_VEL
LIN {X 0,Y 600.369,Z 385.792,A -85,B 0,C 180,E1 28909.889,E2 28909.889} C_VEL
LIN {X 0,Y 600.334,Z 404.158,A -85,B 0,C 180,E1 28909.468,E2 28909.468} C_VEL
LIN {X 0,Y 600.289,Z 421.598,A -85,B 0,C 180,E1 28908.901,E2 28908.901} C_VEL
LIN {X 0,Y 600.23,Z 439.174,A -85,B 0,C 180,E1 28908.149,E2 28908.149} C_VEL
LIN {X 0,Y 600.178,Z 455.879,A -85,B 0,C 180,E1 28907.249,E2 28907.249} C_VEL
LIN {X 0,Y 600.121,Z 471.712,A -85,B 0,C 180,E1 28906.204,E2 28906.204} C_VEL
LIN {X 0,Y 600.066,Z 486.622,A -85,B 0,C 180,E1 28905.016,E2 28905.016} C_VEL
LIN {X 0,Y 600.023,Z 500.529,A -85,B 0,C 180,E1 28903.687,E2 28903.687} C_VEL
LIN {X 0,Y 599.982,Z 513.332,A -85,B 0,C 180,E1 28902.218,E2 28902.218} C_VEL
LIN {X 0,Y 599.951,Z 524.574,A -85,B 0,C 180,E1 28900.66,E2 28900.66} C_VEL
LIN {X 0,Y 599.938,Z 534.271,A -85,B 0,C 180,E1 28899.012,E2 28899.012} C_VEL
LIN {X 0,Y 599.921,Z 541.992,A -85,B 0,C 180,E1 28897.373,E2 28897.373} C_VEL
LIN {X 0,Y 599.913,Z 548.271,A -85,B 0,C 180,E1 28895.643,E2 28895.643} C_VEL
LIN {X 0,Y 599.919,Z 552.779,A -85,B 0,C 180,E1 28893.918,E2 28893.918} C_VEL
LIN {X 0,Y 599.917,Z 555.736,A -85,B 0,C 180,E1 28892.101,E2 28892.101} C_VEL
LIN {X 0,Y 599.909,Z 556.929,A -85,B 0,C 180,E1 28890.286,E2 28890.286} C_VEL
LIN {X 0,Y 599.915,Z 556.379,A -85,B 0,C 180,E1 28888.471,E2 28888.471} C_VEL
LIN {X 0,Y 599.908,Z 554.079,A -85,B 0,C 180,E1 28886.655,E2 28886.655} C_VEL
LIN {X 0,Y 599.914,Z 550.214,A -85,B 0,C 180,E1 28884.932,E2 28884.932} C_VEL
LIN {X 0,Y 599.919,Z 544.63,A -85,B 0,C 180,E1 28883.204,E2 28883.204} C_VEL
LIN {X 0,Y 599.929,Z 537.635,A -85,B 0,C 180,E1 28881.566,E2 28881.566} C_VEL
LIN {X 0,Y 599.948,Z 528.774,A -85,B 0,C 180,E1 28879.921,E2 28879.921} C_VEL
LIN {X 0,Y 599.968,Z 518.467,A -85,B 0,C 180,E1 28878.366,E2 28878.366} C_VEL
LIN {X 0,Y 600.003,Z 506.731,A -85,B 0,C 180,E1 28876.901,E2 28876.901} C_VEL
LIN {X 0,Y 600.04,Z 493.26,A -85,B 0,C 180,E1 28875.497,E2 28875.497} C_VEL
LIN {X 0,Y 600.097,Z 478.778,A -85,B 0,C 180,E1 28874.241,E2 28874.241} C_VEL
LIN {X 0,Y 600.16,Z 462.917,A -85,B 0,C 180,E1 28873.099,E2 28873.099} C_VEL
LIN {X 0,Y 600.218,Z 445.918,A -85,B 0,C 180,E1 28872.1,E2 28872.1} C_VEL
LIN {X 0,Y 600.274,Z 428.802,A -85,B 0,C 180,E1 28871.293,E2 28871.293} C_VEL
LIN {X 0,Y 600.329,Z 410.276,A -85,B 0,C 180,E1 28870.621,E2 28870.621} C_VEL
LIN {X 0,Y 600.362,Z 391.628,A -85,B 0,C 180,E1 28870.135,E2 28870.135} C_VEL
LIN {X 0,Y 600.385,Z 371.886,A -85,B 0,C 180,E1 28869.812,E2 28869.812} C_VEL
LIN {X 0,Y 600.38,Z 175.938,A -85,B 0,C 180,E1 28867.346,E2 28867.346} C_VEL
LIN {X 0,Y 600.302,Z 173.022,A -85,B 0,C 180,E1 28867.164,E2 28867.164} C_VEL
LIN {X 0,Y 600.385,Z 130.91,A -85,B 0,C 180,E1 28864.024,E2 28864.024} C_VEL
LIN {X 0,Y 600.468,Z 96.771,A -85,B 0,C 180,E1 28861.417,E2 28861.417} C_VEL
LIN {X 0,Y 599.972,Z 94.75,A -85,B 0,C 180,E1 28861.208,E2 28861.208} C_VEL
LIN {X 0,Y 599.902,Z 94.755,A -85,B 0,C 180,E1 28858.106,E2 28858.106} C_VEL
LIN {X 0,Y 599.956,Z 94.751,A -85,B 0,C 180,E1 28855.019,E2 28855.019} C_VEL
LIN {X 0,Y 599.943,Z 94.753,A -85,B 0,C 180,E1 28851.928,E2 28851.928} C_VEL
LIN {X 0,Y 599.938,Z 94.749,A -85,B 0,C 180,E1 28848.702,E2 28848.702} C_VEL
LIN {X 0,Y 599.971,Z 94.749,A -85,B 0,C 180,E1 28845.578,E2 28845.578} C_VEL
LIN {X 0,Y 599.957,Z 94.751,A -85,B 0,C 180,E1 28842.414,E2 28842.414} C_VEL
LIN {X 0,Y 599.972,Z 94.745,A -85,B 0,C 180,E1 28839.169,E2 28839.169} C_VEL
LIN {X 0,Y 599.953,Z 94.75,A -85,B 0,C 180,E1 28835.908,E2 28835.908} C_VEL
LIN {X 0,Y 599.977,Z 94.753,A -85,B 0,C 180,E1 28832.68,E2 28832.68} C_VEL
LIN {X 0,Y 599.964,Z 94.748,A -85,B 0,C 180,E1 28829.448,E2 28829.448} C_VEL
LIN {X 0,Y 599.975,Z 94.833,A -85,B 0,C 180,E1 28828.669,E2 28828.669} C_VEL
LIN {X 0,Y 600.492,Z 98.164,A -85,B 0,C 180,E1 28828.384,E2 28828.384} C_VEL
LIN {X 0,Y 600.416,Z 138.14,A -85,B 0,C 180,E1 28825.339,E2 28825.339} C_VEL
LIN {X 0,Y 600.306,Z 175.732,A -85,B 0,C 180,E1 28822.57,E2 28822.57} C_VEL
LIN {X 0,Y 600.365,Z 328.807,A -85,B 0,C 180,E1 28820.637,E2 28820.637} C_VEL
LIN {X 0,Y 600.374,Z 385.148,A -85,B 0,C 180,E1 28819.902,E2 28819.902} C_VEL
LIN {X 0,Y 600.339,Z 404.191,A -85,B 0,C 180,E1 28819.468,E2 28819.468} C_VEL
LIN {X 0,Y 600.282,Z 422.808,A -85,B 0,C 180,E1 28818.853,E2 28818.853} C_VEL
LIN {X 0,Y 600.231,Z 440.144,A -85,B 0,C 180,E1 28818.102,E2 28818.102} C_VEL
LIN {X 0,Y 600.174,Z 457.483,A -85,B 0,C 180,E1 28817.15,E2 28817.15} C_VEL
LIN {X 0,Y 600.114,Z 473.688,A -85,B 0,C 180,E1 28816.056,E2 28816.056} C_VEL
LIN {X 0,Y 600.06,Z 488.821,A -85,B 0,C 180,E1 28814.82,E2 28814.82} C_VEL
LIN {X 0,Y 600.013,Z 503.309,A -85,B 0,C 180,E1 28813.393,E2 28813.393} C_VEL
LIN {X 0,Y 599.979,Z 515.638,A -85,B 0,C 180,E1 28811.926,E2 28811.926} C_VEL
LIN {X 0,Y 599.956,Z 526.482,A -85,B 0,C 180,E1 28810.369,E2 28810.369} C_VEL
LIN {X 0,Y 599.934,Z 535.805,A -85,B 0,C 180,E1 28808.723,E2 28808.723} C_VEL
LIN {X 0,Y 599.918,Z 543.584,A -85,B 0,C 180,E1 28806.988,E2 28806.988} C_VEL
LIN {X 0,Y 599.916,Z 549.462,A -85,B 0,C 180,E1 28805.26,E2 28805.26} C_VEL
LIN {X 0,Y 599.912,Z 553.766,A -85,B 0,C 180,E1 28803.44,E2 28803.44} C_VEL
LIN {X 0,Y 599.911,Z 556.255,A -85,B 0,C 180,E1 28801.624,E2 28801.624} C_VEL
LIN {X 0,Y 599.912,Z 556.97,A -85,B 0,C 180,E1 28799.809,E2 28799.809} C_VEL
LIN {X 0,Y 599.905,Z 555.955,A -85,B 0,C 180,E1 28797.994,E2 28797.994} C_VEL
LIN {X 0,Y 599.916,Z 553.175,A -85,B 0,C 180,E1 28796.178,E2 28796.178} C_VEL
LIN {X 0,Y 599.918,Z 548.858,A -85,B 0,C 180,E1 28794.453,E2 28794.453} C_VEL
LIN {X 0,Y 599.921,Z 542.778,A -85,B 0,C 180,E1 28792.723,E2 28792.723} C_VEL
LIN {X 0,Y 599.932,Z 535.267,A -85,B 0,C 180,E1 28791.084,E2 28791.084} C_VEL
LIN {X 0,Y 599.954,Z 525.806,A -85,B 0,C 180,E1 28789.437,E2 28789.437} C_VEL
LIN {X 0,Y 599.983,Z 514.814,A -85,B 0,C 180,E1 28787.879,E2 28787.879} C_VEL
LIN {X 0,Y 600.02,Z 502.31,A -85,B 0,C 180,E1 28786.411,E2 28786.411} C_VEL
LIN {X 0,Y 600.062,Z 488.164,A -85,B 0,C 180,E1 28785.033,E2 28785.033} C_VEL
LIN {X 0,Y 600.117,Z 472.917,A -85,B 0,C 180,E1 28783.795,E2 28783.795} C_VEL
LIN {X 0,Y 600.173,Z 457.316,A -85,B 0,C 180,E1 28782.75,E2 28782.75} C_VEL
LIN {X 0,Y 600.231,Z 439.983,A -85,B 0,C 180,E1 28781.8,E2 28781.8} C_VEL
LIN {X 0,Y 600.283,Z 422.557,A -85,B 0,C 180,E1 28781.047,E2 28781.047} C_VEL
LIN {X 0,Y 600.334,Z 404.009,A -85,B 0,C 180,E1 28780.438,E2 28780.438} C_VEL
LIN {X 0,Y 600.375,Z 384.909,A -85,B 0,C 180,E1 28780.003,E2 28780.003} C_VEL
LIN {X 0,Y 600.405,Z 311.523,A -85,B 0,C 180,E1 28779.057,E2 28779.057} C_VEL
LIN {X 0,Y 600.311,Z 175.246,A -85,B 0,C 180,E1 28777.329,E2 28777.329} C_VEL
LIN {X 0,Y 600.407,Z 133.025,A -85,B 0,C 180,E1 28774.185,E2 28774.185} C_VEL
LIN {X 0,Y 600.542,Z 96.877,A -85,B 0,C 180,E1 28771.429,E2 28771.429} C_VEL
LIN {X 0,Y 599.976,Z 94.754,A -85,B 0,C 180,E1 28771.209,E2 28771.209} C_VEL
LIN {X 0,Y 599.945,Z 94.749,A -85,B 0,C 180,E1 28768.027,E2 28768.027} C_VEL
LIN {X 0,Y 599.931,Z 94.752,A -85,B 0,C 180,E1 28764.751,E2 28764.751} C_VEL
LIN {X 0,Y 599.972,Z 94.75,A -85,B 0,C 180,E1 28761.688,E2 28761.688} C_VEL
LIN {X 0,Y 599.911,Z 94.752,A -85,B 0,C 180,E1 28758.573,E2 28758.573} C_VEL
LIN {X 0,Y 599.954,Z 94.754,A -85,B 0,C 180,E1 28755.443,E2 28755.443} C_VEL
LIN {X 0,Y 599.9,Z 94.754,A -85,B 0,C 180,E1 28752.55,E2 28752.55} C_VEL
LIN {X 0,Y 599.921,Z 94.754,A -85,B 0,C 180,E1 28749.347,E2 28749.347} C_VEL
LIN {X 0,Y 599.914,Z 94.754,A -85,B 0,C 180,E1 28746.513,E2 28746.513} C_VEL
LIN {X 0,Y 599.919,Z 94.753,A -85,B 0,C 180,E1 28743.211,E2 28743.211} C_VEL
LIN {X 0,Y 599.969,Z 94.854,A -85,B 0,C 180,E1 28742.256,E2 28742.256} C_VEL
LIN {X 0,Y 600.805,Z 98.009,A -85,B 0,C 180,E1 28742.009,E2 28742.009} C_VEL
LIN {X 0,Y 600.653,Z 147.597,A -85,B 0,C 180,E1 28738.974,E2 28738.974} C_VEL
LIN {X 0,Y 600.706,Z 163.43,A -85,B 0,C 180,E1 28738.044,E2 28738.044} C_VEL
LIN {X 0,Y 600.661,Z 367.83,A -85,B 0,C 180,E1 28735.367,E2 28735.367} C_VEL
LIN {X 0,Y 600.611,Z 426.191,A -85,B 0,C 180,E1 28734.585,E2 28734.585} C_VEL
LIN {X 0,Y 600.568,Z 446.685,A -85,B 0,C 180,E1 28734.125,E2 28734.125} C_VEL
LIN {X 0,Y 600.501,Z 465.761,A -85,B 0,C 180,E1 28733.528,E2 28733.528} C_VEL
LIN {X 0,Y 600.421,Z 485.597,A -85,B 0,C 180,E1 28732.728,E2 28732.728} C_VEL
LIN {X 0,Y 600.349,Z 504.044,A -85,B 0,C 180,E1 28731.802,E2 28731.802} C_VEL
LIN {X 0,Y 600.277,Z 522.523,A -85,B 0,C 180,E1 28730.679,E2 28730.679} C_VEL
LIN {X 0,Y 600.197,Z 540.561,A -85,B 0,C 180,E1 28729.361,E2 28729.361} C_VEL
LIN {X 0,Y 600.126,Z 557.359,A -85,B 0,C 180,E1 28727.903,E2 28727.903} C_VEL
LIN {X 0,Y 600.055,Z 572.905,A -85,B 0,C 180,E1 28726.307,E2 28726.307} C_VEL
LIN {X 0,Y 600.01,Z 587.128,A -85,B 0,C 180,E1 28724.574,E2 28724.574} C_VEL
LIN {X 0,Y 599.969,Z 599.291,A -85,B 0,C 180,E1 28722.806,E2 28722.806} C_VEL
LIN {X 0,Y 599.948,Z 609.598,A -85,B 0,C 180,E1 28721.005,E2 28721.005} C_VEL
LIN {X 0,Y 599.928,Z 618.058,A -85,B 0,C 180,E1 28719.207,E2 28719.207} C_VEL
LIN {X 0,Y 599.915,Z 624.989,A -85,B 0,C 180,E1 28717.374,E2 28717.374} C_VEL
LIN {X 0,Y 599.909,Z 630.506,A -85,B 0,C 180,E1 28715.452,E2 28715.452} C_VEL
LIN {X 0,Y 599.905,Z 634.239,A -85,B 0,C 180,E1 28713.536,E2 28713.536} C_VEL
LIN {X 0,Y 599.904,Z 636.372,A -85,B 0,C 180,E1 28711.624,E2 28711.624} C_VEL
LIN {X 0,Y 599.9,Z 636.918,A -85,B 0,C 180,E1 28709.619,E2 28709.619} C_VEL
LIN {X 0,Y 599.901,Z 635.839,A -85,B 0,C 180,E1 28707.708,E2 28707.708} C_VEL
LIN {X 0,Y 599.905,Z 633.136,A -85,B 0,C 180,E1 28705.795,E2 28705.795} C_VEL
LIN {X 0,Y 599.91,Z 628.737,A -85,B 0,C 180,E1 28703.877,E2 28703.877} C_VEL
LIN {X 0,Y 599.92,Z 622.621,A -85,B 0,C 180,E1 28701.953,E2 28701.953} C_VEL
LIN {X 0,Y 599.932,Z 614.805,A -85,B 0,C 180,E1 28700.054,E2 28700.054} C_VEL
LIN {X 0,Y 599.946,Z 605.72,A -85,B 0,C 180,E1 28698.269,E2 28698.269} C_VEL
LIN {X 0,Y 599.975,Z 594.82,A -85,B 0,C 180,E1 28696.509,E2 28696.509} C_VEL
LIN {X 0,Y 600.021,Z 582.491,A -85,B 0,C 180,E1 28694.834,E2 28694.834} C_VEL
LIN {X 0,Y 600.069,Z 568.748,A -85,B 0,C 180,E1 28693.247,E2 28693.247} C_VEL
LIN {X 0,Y 600.132,Z 553.446,A -85,B 0,C 180,E1 28691.742,E2 28691.742} C_VEL
LIN {X 0,Y 600.207,Z 536.616,A -85,B 0,C 180,E1 28690.337,E2 28690.337} C_VEL
LIN {X 0,Y 600.29,Z 519.362,A -85,B 0,C 180,E1 28689.119,E2 28689.119} C_VEL
LIN {X 0,Y 600.374,Z 501.265,A -85,B 0,C 180,E1 28688.046,E2 28688.046} C_VEL
LIN {X 0,Y 600.441,Z 482.254,A -85,B 0,C 180,E1 28687.119,E2 28687.119} C_VEL
LIN {X 0,Y 600.507,Z 462.86,A -85,B 0,C 180,E1 28686.369,E2 28686.369} C_VEL
LIN {X 0,Y 600.573,Z 442.716,A -85,B 0,C 180,E1 28685.775,E2 28685.775} C_VEL
LIN {X 0,Y 600.617,Z 422.202,A -85,B 0,C 180,E1 28685.352,E2 28685.352} C_VEL
LIN {X 0,Y 600.818,Z 171.659,A -85,B 0,C 180,E1 28682.07,E2 28682.07} C_VEL
LIN {X 0,Y 600.618,Z 162.84,A -85,B 0,C 180,E1 28681.942,E2 28681.942} C_VEL
LIN {X 0,Y 600.712,Z 113.36,A -85,B 0,C 180,E1 28678.938,E2 28678.938} C_VEL
LIN {X 0,Y 600.63,Z 97.066,A -85,B 0,C 180,E1 28677.922,E2 28677.922} C_VEL
LIN {X 0,Y 599.959,Z 94.755,A -85,B 0,C 180,E1 28677.716,E2 28677.716} C_VEL
LIN {X 0,Y 599.928,Z 94.751,A -85,B 0,C 180,E1 28674.668,E2 28674.668} C_VEL
LIN {X 0,Y 599.925,Z 94.752,A -85,B 0,C 180,E1 28671.412,E2 28671.412} C_VEL
LIN {X 0,Y 599.952,Z 94.749,A -85,B 0,C 180,E1 28668.442,E2 28668.442} C_VEL
LIN {X 0,Y 599.916,Z 94.752,A -85,B 0,C 180,E1 28665.306,E2 28665.306} C_VEL
LIN {X 0,Y 599.975,Z 94.749,A -85,B 0,C 180,E1 28662.276,E2 28662.276} C_VEL
LIN {X 0,Y 599.911,Z 94.749,A -85,B 0,C 180,E1 28659.173,E2 28659.173} C_VEL
LIN {X 0,Y 599.975,Z 94.754,A -85,B 0,C 180,E1 28656.034,E2 28656.034} C_VEL
LIN {X 0,Y 599.913,Z 94.75,A -85,B 0,C 180,E1 28653.025,E2 28653.025} C_VEL
LIN {X 0,Y 599.95,Z 94.753,A -85,B 0,C 180,E1 28649.888,E2 28649.888} C_VEL
LIN {X 0,Y 599.918,Z 94.751,A -85,B 0,C 180,E1 28646.919,E2 28646.919} C_VEL
LIN {X 0,Y 599.917,Z 94.752,A -85,B 0,C 180,E1 28643.578,E2 28643.578} C_VEL
LIN {X 0,Y 599.938,Z 94.751,A -85,B 0,C 180,E1 28640.69,E2 28640.69} C_VEL
LIN {X 0,Y 599.912,Z 94.752,A -85,B 0,C 180,E1 28637.558,E2 28637.558} C_VEL
LIN {X 0,Y 599.972,Z 94.75,A -85,B 0,C 180,E1 28634.476,E2 28634.476} C_VEL
LIN {X 0,Y 599.905,Z 94.752,A -85,B 0,C 180,E1 28631.44,E2 28631.44} C_VEL
LIN {X 0,Y 599.973,Z 94.752,A -85,B 0,C 180,E1 28628.433,E2 28628.433} C_VEL
LIN {X 0,Y 599.903,Z 94.752,A -85,B 0,C 180,E1 28625.355,E2 28625.355} C_VEL
LIN {X 0,Y 599.969,Z 94.753,A -85,B 0,C 180,E1 28622.292,E2 28622.292} C_VEL
LIN {X 0,Y 599.902,Z 94.752,A -85,B 0,C 180,E1 28619.331,E2 28619.331} C_VEL
LIN {X 0,Y 599.945,Z 94.753,A -85,B 0,C 180,E1 28616.177,E2 28616.177} C_VEL
LIN {X 0,Y 599.9,Z 94.752,A -85,B 0,C 180,E1 28613.45,E2 28613.45} C_VEL
LIN {X 0,Y 598.933,Z 94.879,A -85,B 0,C 180,E1 28612.714,E2 28612.714} C_VEL
LIN {X 0,Y 592.466,Z 95.688,A -85,B 0,C 180,E1 28610.596,E2 28610.596} C_VEL
LIN {X 0,Y 591.994,Z 95.741,A -85,B 0,C 180,E1 28610.113,E2 28610.113} C_VEL
LIN {X 0,Y 591.968,Z 95.74,A -85,B 0,C 180,E1 28607.216,E2 28607.216} C_VEL
LIN {X 0,Y 591.97,Z 95.742,A -85,B 0,C 180,E1 28603.918,E2 28603.918} C_VEL
LIN {X 0,Y 591.99,Z 95.74,A -85,B 0,C 180,E1 28600.975,E2 28600.975} C_VEL
LIN {X 0,Y 591.961,Z 95.741,A -85,B 0,C 180,E1 28597.768,E2 28597.768} C_VEL
LIN {X 0,Y 592.027,Z 95.741,A -85,B 0,C 180,E1 28594.704,E2 28594.704} C_VEL
LIN {X 0,Y 591.957,Z 95.74,A -85,B 0,C 180,E1 28591.641,E2 28591.641} C_VEL
LIN {X 0,Y 592.022,Z 95.742,A -85,B 0,C 180,E1 28588.525,E2 28588.525} C_VEL
LIN {X 0,Y 591.96,Z 95.742,A -85,B 0,C 180,E1 28585.422,E2 28585.422} C_VEL
LIN {X 0,Y 591.974,Z 95.743,A -85,B 0,C 180,E1 28582.185,E2 28582.185} C_VEL
LIN {X 0,Y 591.968,Z 95.742,A -85,B 0,C 180,E1 28579.309,E2 28579.309} C_VEL
LIN {X 0,Y 591.959,Z 95.742,A -85,B 0,C 180,E1 28576.015,E2 28576.015} C_VEL
LIN {X 0,Y 591.987,Z 95.743,A -85,B 0,C 180,E1 28573.143,E2 28573.143} C_VEL
LIN {X 0,Y 591.959,Z 95.743,A -85,B 0,C 180,E1 28570.055,E2 28570.055} C_VEL
LIN {X 0,Y 591.993,Z 95.743,A -85,B 0,C 180,E1 28567.137,E2 28567.137} C_VEL
LIN {X 0,Y 591.956,Z 95.744,A -85,B 0,C 180,E1 28563.969,E2 28563.969} C_VEL
LIN {X 0,Y 592.031,Z 95.744,A -85,B 0,C 180,E1 28560.913,E2 28560.913} C_VEL
LIN {X 0,Y 592.033,Z 95.863,A -85,B 0,C 180,E1 28559.029,E2 28559.029} C_VEL
LIN {X 0,Y 593.116,Z 100.407,A -85,B 0,C 180,E1 28558.604,E2 28558.604} C_VEL
LIN {X 0,Y 592.916,Z 138.164,A -85,B 0,C 180,E1 28555.682,E2 28555.682} C_VEL
LIN {X 0,Y 592.772,Z 175.819,A -85,B 0,C 180,E1 28552.872,E2 28552.872} C_VEL
LIN {X 0,Y 593.08,Z 182.688,A -85,B 0,C 180,E1 28552.771,E2 28552.771} C_VEL
LIN {X 0,Y 592.847,Z 384.364,A -85,B 0,C 180,E1 28550.181,E2 28550.181} C_VEL
LIN {X 0,Y 592.77,Z 403.331,A -85,B 0,C 180,E1 28549.751,E2 28549.751} C_VEL
LIN {X 0,Y 592.684,Z 421.167,A -85,B 0,C 180,E1 28549.17,E2 28549.17} C_VEL
LIN {X 0,Y 592.563,Z 439.182,A -85,B 0,C 180,E1 28548.392,E2 28548.392} C_VEL
LIN {X 0,Y 592.455,Z 455.885,A -85,B 0,C 180,E1 28547.481,E2 28547.481} C_VEL
LIN {X 0,Y 592.339,Z 471.718,A -85,B 0,C 180,E1 28546.423,E2 28546.423} C_VEL
LIN {X 0,Y 592.229,Z 486.627,A -85,B 0,C 180,E1 28545.22,E2 28545.22} C_VEL
LIN {X 0,Y 592.129,Z 500.534,A -85,B 0,C 180,E1 28543.873,E2 28543.873} C_VEL
LIN {X 0,Y 592.052,Z 513.339,A -85,B 0,C 180,E1 28542.384,E2 28542.384} C_VEL
LIN {X 0,Y 591.996,Z 524.579,A -85,B 0,C 180,E1 28540.805,E2 28540.805} C_VEL
LIN {X 0,Y 591.956,Z 534.275,A -85,B 0,C 180,E1 28539.135,E2 28539.135} C_VEL
LIN {X 0,Y 591.933,Z 542.036,A -85,B 0,C 180,E1 28537.463,E2 28537.463} C_VEL
LIN {X 0,Y 591.917,Z 548.274,A -85,B 0,C 180,E1 28535.719,E2 28535.719} C_VEL
LIN {X 0,Y 591.919,Z 552.781,A -85,B 0,C 180,E1 28533.971,E2 28533.971} C_VEL
LIN {X 0,Y 591.917,Z 555.738,A -85,B 0,C 180,E1 28532.129,E2 28532.129} C_VEL
LIN {X 0,Y 591.909,Z 556.929,A -85,B 0,C 180,E1 28530.29,E2 28530.29} C_VEL
LIN {X 0,Y 591.915,Z 556.38,A -85,B 0,C 180,E1 28528.451,E2 28528.451} C_VEL
LIN {X 0,Y 591.908,Z 554.079,A -85,B 0,C 180,E1 28526.61,E2 28526.61} C_VEL
LIN {X 0,Y 591.916,Z 550.213,A -85,B 0,C 180,E1 28524.863,E2 28524.863} C_VEL
LIN {X 0,Y 591.93,Z 544.628,A -85,B 0,C 180,E1 28523.111,E2 28523.111} C_VEL
LIN {X 0,Y 591.941,Z 537.633,A -85,B 0,C 180,E1 28521.451,E2 28521.451} C_VEL
LIN {X 0,Y 591.979,Z 528.772,A -85,B 0,C 180,E1 28519.784,E2 28519.784} C_VEL
LIN {X 0,Y 592.024,Z 518.464,A -85,B 0,C 180,E1 28518.208,E2 28518.208} C_VEL
LIN {X 0,Y 592.093,Z 506.726,A -85,B 0,C 180,E1 28516.722,E2 28516.722} C_VEL
LIN {X 0,Y 592.175,Z 493.536,A -85,B 0,C 180,E1 28515.328,E2 28515.328} C_VEL
LIN {X 0,Y 592.291,Z 478.767,A -85,B 0,C 180,E1 28514.028,E2 28514.028} C_VEL
LIN {X 0,Y 592.413,Z 462.905,A -85,B 0,C 180,E1 28512.871,E2 28512.871} C_VEL
LIN {X 0,Y 592.532,Z 445.91,A -85,B 0,C 180,E1 28511.86,E2 28511.86} C_VEL
LIN {X 0,Y 592.646,Z 428.451,A -85,B 0,C 180,E1 28511.03,E2 28511.03} C_VEL
LIN {X 0,Y 592.751,Z 410.041,A -85,B 0,C 180,E1 28510.357,E2 28510.357} C_VEL
LIN {X 0,Y 592.826,Z 391.433,A -85,B 0,C 180,E1 28509.868,E2 28509.868} C_VEL
LIN {X 0,Y 592.874,Z 371.58,A -85,B 0,C 180,E1 28509.542,E2 28509.542} C_VEL
LIN {X 0,Y 592.987,Z 177.009,A -85,B 0,C 180,E1 28507.062,E2 28507.062} C_VEL
LIN {X 0,Y 592.709,Z 175.035,A -85,B 0,C 180,E1 28507.006,E2 28507.006} C_VEL
LIN {X 0,Y 592.915,Z 132.305,A -85,B 0,C 180,E1 28503.779,E2 28503.779} C_VEL
LIN {X 0,Y 593.118,Z 99.528,A -85,B 0,C 180,E1 28501.235,E2 28501.235} C_VEL
LIN {X 0,Y 592.005,Z 95.743,A -85,B 0,C 180,E1 28500.867,E2 28500.867} C_VEL
LIN {X 0,Y 591.975,Z 95.744,A -85,B 0,C 180,E1 28497.856,E2 28497.856} C_VEL
LIN {X 0,Y 591.982,Z 95.741,A -85,B 0,C 180,E1 28494.596,E2 28494.596} C_VEL
LIN {X 0,Y 592.039,Z 95.738,A -85,B 0,C 180,E1 28491.574,E2 28491.574} C_VEL
LIN {X 0,Y 591.997,Z 95.74,A -85,B 0,C 180,E1 28488.412,E2 28488.412} C_VEL
LIN {X 0,Y 592.033,Z 95.735,A -85,B 0,C 180,E1 28485.18,E2 28485.18} C_VEL
LIN {X 0,Y 592.033,Z 95.741,A -85,B 0,C 180,E1 28481.974,E2 28481.974} C_VEL
LIN {X 0,Y 592.022,Z 95.739,A -85,B 0,C 180,E1 28478.674,E2 28478.674} C_VEL
LIN {X 0,Y 592.032,Z 95.734,A -85,B 0,C 180,E1 28475.4,E2 28475.4} C_VEL
LIN {X 0,Y 592.008,Z 95.741,A -85,B 0,C 180,E1 28472.142,E2 28472.142} C_VEL
LIN {X 0,Y 592.057,Z 95.891,A -85,B 0,C 180,E1 28468.992,E2 28468.992} C_VEL
LIN {X 0,Y 593.105,Z 100.202,A -85,B 0,C 180,E1 28468.605,E2 28468.605} C_VEL
LIN {X 0,Y 592.923,Z 139.848,A -85,B 0,C 180,E1 28465.553,E2 28465.553} C_VEL
LIN {X 0,Y 592.727,Z 175.779,A -85,B 0,C 180,E1 28462.875,E2 28462.875} C_VEL
LIN {X 0,Y 593.055,Z 181.974,A -85,B 0,C 180,E1 28462.781,E2 28462.781} C_VEL
LIN {X 0,Y 592.852,Z 384.519,A -85,B 0,C 180,E1 28460.179,E2 28460.179} C_VEL
LIN {X 0,Y 592.773,Z 403.541,A -85,B 0,C 180,E1 28459.744,E2 28459.744} C_VEL
LIN {X 0,Y 592.666,Z 422.087,A -85,B 0,C 180,E1 28459.134,E2 28459.134} C_VEL
LIN {X 0,Y 592.562,Z 439.902,A -85,B 0,C 180,E1 28458.358,E2 28458.358} C_VEL
LIN {X 0,Y 592.44,Z 457.498,A -85,B 0,C 180,E1 28457.381,E2 28457.381} C_VEL
LIN {X 0,Y 592.316,Z 474.361,A -85,B 0,C 180,E1 28456.223,E2 28456.223} C_VEL
LIN {X 0,Y 592.21,Z 489.383,A -85,B 0,C 180,E1 28454.97,E2 28454.97} C_VEL
LIN {X 0,Y 592.119,Z 503.32,A -85,B 0,C 180,E1 28453.575,E2 28453.575} C_VEL
LIN {X 0,Y 592.046,Z 515.649,A -85,B 0,C 180,E1 28452.087,E2 28452.087} C_VEL
LIN {X 0,Y 591.996,Z 526.477,A -85,B 0,C 180,E1 28450.51,E2 28450.51} C_VEL
LIN {X 0,Y 591.955,Z 535.802,A -85,B 0,C 180,E1 28448.842,E2 28448.842} C_VEL
LIN {X 0,Y 591.924,Z 543.579,A -85,B 0,C 180,E1 28447.083,E2 28447.083} C_VEL
LIN {X 0,Y 591.921,Z 549.457,A -85,B 0,C 180,E1 28445.331,E2 28445.331} C_VEL
LIN {X 0,Y 591.912,Z 553.761,A -85,B 0,C 180,E1 28443.487,E2 28443.487} C_VEL
LIN {X 0,Y 591.91,Z 556.256,A -85,B 0,C 180,E1 28441.646,E2 28441.646} C_VEL
LIN {X 0,Y 591.912,Z 556.968,A -85,B 0,C 180,E1 28439.807,E2 28439.807} C_VEL
LIN {X 0,Y 591.905,Z 555.959,A -85,B 0,C 180,E1 28437.967,E2 28437.967} C_VEL
LIN {X 0,Y 591.916,Z 553.175,A -85,B 0,C 180,E1 28436.126,E2 28436.126} C_VEL
LIN {X 0,Y 591.918,Z 548.859,A -85,B 0,C 180,E1 28434.378,E2 28434.378} C_VEL
LIN {X 0,Y 591.931,Z 542.778,A -85,B 0,C 180,E1 28432.624,E2 28432.624} C_VEL
LIN {X 0,Y 591.956,Z 535.255,A -85,B 0,C 180,E1 28430.963,E2 28430.963} C_VEL
LIN {X 0,Y 591.993,Z 525.806,A -85,B 0,C 180,E1 28429.293,E2 28429.293} C_VEL
LIN {X 0,Y 592.051,Z 514.804,A -85,B 0,C 180,E1 28427.714,E2 28427.714} C_VEL
LIN {X 0,Y 592.126,Z 502.311,A -85,B 0,C 180,E1 28426.226,E2 28426.226} C_VEL
LIN {X 0,Y 592.215,Z 488.153,A -85,B 0,C 180,E1 28424.83,E2 28424.83} C_VEL
LIN {X 0,Y 592.328,Z 472.917,A -85,B 0,C 180,E1 28423.576,E2 28423.576} C_VEL
LIN {X 0,Y 592.437,Z 457.298,A -85,B 0,C 180,E1 28422.518,E2 28422.518} C_VEL
LIN {X 0,Y 592.565,Z 439.983,A -85,B 0,C 180,E1 28421.556,E2 28421.556} C_VEL
LIN {X 0,Y 592.664,Z 422.543,A -85,B 0,C 180,E1 28420.794,E2 28420.794} C_VEL
LIN {X 0,Y 592.765,Z 403.945,A -85,B 0,C 180,E1 28420.177,E2 28420.177} C_VEL
LIN {X 0,Y 592.848,Z 384.893,A -85,B 0,C 180,E1 28419.738,E2 28419.738} C_VEL
LIN {X 0,Y 592.938,Z 298.582,A -85,B 0,C 180,E1 28418.617,E2 28418.617} C_VEL
LIN {X 0,Y 592.915,Z 176.526,A -85,B 0,C 180,E1 28417.053,E2 28417.053} C_VEL
LIN {X 0,Y 592.717,Z 175.098,A -85,B 0,C 180,E1 28417.011,E2 28417.011} C_VEL
LIN {X 0,Y 592.934,Z 133.718,A -85,B 0,C 180,E1 28413.889,E2 28413.889} C_VEL
LIN {X 0,Y 593.044,Z 99.362,A -85,B 0,C 180,E1 28411.248,E2 28411.248} C_VEL
LIN {X 0,Y 592.025,Z 95.744,A -85,B 0,C 180,E1 28410.942,E2 28410.942} C_VEL
LIN {X 0,Y 592.029,Z 95.737,A -85,B 0,C 180,E1 28407.746,E2 28407.746} C_VEL
LIN {X 0,Y 591.987,Z 95.741,A -85,B 0,C 180,E1 28404.597,E2 28404.597} C_VEL
LIN {X 0,Y 592.032,Z 95.744,A -85,B 0,C 180,E1 28401.439,E2 28401.439} C_VEL
LIN {X 0,Y 591.976,Z 95.741,A -85,B 0,C 180,E1 28398.411,E2 28398.411} C_VEL
LIN {X 0,Y 591.986,Z 95.743,A -85,B 0,C 180,E1 28395.185,E2 28395.185} C_VEL
LIN {X 0,Y 591.975,Z 95.743,A -85,B 0,C 180,E1 28392.287,E2 28392.287} C_VEL
LIN {X 0,Y 591.961,Z 95.744,A -85,B 0,C 180,E1 28389.016,E2 28389.016} C_VEL
LIN {X 0,Y 592.029,Z 95.744,A -85,B 0,C 180,E1 28385.996,E2 28385.996} C_VEL
LIN {X 0,Y 591.975,Z 95.745,A -85,B 0,C 180,E1 28382.832,E2 28382.832} C_VEL
LIN {X 0,Y 591.981,Z 95.756,A -85,B 0,C 180,E1 28382.688,E2 28382.688} C_VEL
LIN {X 0,Y 593.716,Z 100.714,A -85,B 0,C 180,E1 28382.266,E2 28382.266} C_VEL
LIN {X 0,Y 593.405,Z 150.301,A -85,B 0,C 180,E1 28379.196,E2 28379.196} C_VEL
LIN {X 0,Y 593.436,Z 163.477,A -85,B 0,C 180,E1 28378.418,E2 28378.418} C_VEL
LIN {X 0,Y 593.755,Z 169.468,A -85,B 0,C 180,E1 28378.321,E2 28378.321} C_VEL
LIN {X 0,Y 593.363,Z 409.443,A -85,B 0,C 180,E1 28375.155,E2 28375.155} C_VEL
LIN {X 0,Y 593.304,Z 431.789,A -85,B 0,C 180,E1 28374.793,E2 28374.793} C_VEL
LIN {X 0,Y 593.188,Z 452.329,A -85,B 0,C 180,E1 28374.281,E2 28374.281} C_VEL
LIN {X 0,Y 593.08,Z 470.852,A -85,B 0,C 180,E1 28373.656,E2 28373.656} C_VEL
LIN {X 0,Y 592.922,Z 490.076,A -85,B 0,C 180,E1 28372.822,E2 28372.822} C_VEL
LIN {X 0,Y 592.768,Z 508.503,A -85,B 0,C 180,E1 28371.835,E2 28371.835} C_VEL
LIN {X 0,Y 592.598,Z 526.903,A -85,B 0,C 180,E1 28370.649,E2 28370.649} C_VEL
LIN {X 0,Y 592.437,Z 544.213,A -85,B 0,C 180,E1 28369.317,E2 28369.317} C_VEL
LIN {X 0,Y 592.302,Z 559.92,A -85,B 0,C 180,E1 28367.893,E2 28367.893} C_VEL
LIN {X 0,Y 592.189,Z 574.197,A -85,B 0,C 180,E1 28366.378,E2 28366.378} C_VEL
LIN {X 0,Y 592.1,Z 587.852,A -85,B 0,C 180,E1 28364.673,E2 28364.673} C_VEL
LIN {X 0,Y 592.027,Z 599.924,A -85,B 0,C 180,E1 28362.882,E2 28362.882} C_VEL
LIN {X 0,Y 591.978,Z 610.395,A -85,B 0,C 180,E1 28361.003,E2 28361.003} C_VEL
LIN {X 0,Y 591.943,Z 618.871,A -85,B 0,C 180,E1 28359.136,E2 28359.136} C_VEL
LIN {X 0,Y 591.921,Z 625.897,A -85,B 0,C 180,E1 28357.181,E2 28357.181} C_VEL
LIN {X 0,Y 591.91,Z 631.142,A -85,B 0,C 180,E1 28355.234,E2 28355.234} C_VEL
LIN {X 0,Y 591.905,Z 634.709,A -85,B 0,C 180,E1 28353.293,E2 28353.293} C_VEL
LIN {X 0,Y 591.904,Z 636.639,A -85,B 0,C 180,E1 28351.259,E2 28351.259} C_VEL
LIN {X 0,Y 591.903,Z 636.852,A -85,B 0,C 180,E1 28349.323,E2 28349.323} C_VEL
LIN {X 0,Y 591.909,Z 635.392,A -85,B 0,C 180,E1 28347.29,E2 28347.29} C_VEL
LIN {X 0,Y 591.915,Z 632.17,A -85,B 0,C 180,E1 28345.253,E2 28345.253} C_VEL
LIN {X 0,Y 591.925,Z 627.416,A -85,B 0,C 180,E1 28343.308,E2 28343.308} C_VEL
LIN {X 0,Y 591.94,Z 620.853,A -85,B 0,C 180,E1 28341.355,E2 28341.355} C_VEL
LIN {X 0,Y 591.961,Z 612.796,A -85,B 0,C 180,E1 28339.49,E2 28339.49} C_VEL
LIN {X 0,Y 591.999,Z 602.839,A -85,B 0,C 180,E1 28337.615,E2 28337.615} C_VEL
LIN {X 0,Y 592.07,Z 591.03,A -85,B 0,C 180,E1 28335.775,E2 28335.775} C_VEL
LIN {X 0,Y 592.164,Z 578.452,A -85,B 0,C 180,E1 28334.126,E2 28334.126} C_VEL
LIN {X 0,Y 592.277,Z 563.98,A -85,B 0,C 180,E1 28332.514,E2 28332.514} C_VEL
LIN {X 0,Y 592.417,Z 548.451,A -85,B 0,C 180,E1 28331.042,E2 28331.042} C_VEL
LIN {X 0,Y 592.575,Z 531.281,A -85,B 0,C 180,E1 28329.661,E2 28329.661} C_VEL
LIN {X 0,Y 592.737,Z 512.921,A -85,B 0,C 180,E1 28328.425,E2 28328.425} C_VEL
LIN {X 0,Y 592.869,Z 494.305,A -85,B 0,C 180,E1 28327.387,E2 28327.387} C_VEL
LIN {X 0,Y 593.034,Z 475.126,A -85,B 0,C 180,E1 28326.518,E2 28326.518} C_VEL
LIN {X 0,Y 593.181,Z 454.593,A -85,B 0,C 180,E1 28325.788,E2 28325.788} C_VEL
LIN {X 0,Y 593.297,Z 434.572,A -85,B 0,C 180,E1 28325.264,E2 28325.264} C_VEL
LIN {X 0,Y 593.358,Z 413.994,A -85,B 0,C 180,E1 28324.905,E2 28324.905} C_VEL
LIN {X 0,Y 593.738,Z 175.552,A -85,B 0,C 180,E1 28321.76,E2 28321.76} C_VEL
LIN {X 0,Y 593.537,Z 164.076,A -85,B 0,C 180,E1 28321.595,E2 28321.595} C_VEL
LIN {X 0,Y 593.343,Z 162.045,A -85,B 0,C 180,E1 28321.518,E2 28321.518} C_VEL
LIN {X 0,Y 593.591,Z 113.36,A -85,B 0,C 180,E1 28318.523,E2 28318.523} C_VEL
LIN {X 0,Y 593.679,Z 100.545,A -85,B 0,C 180,E1 28317.721,E2 28317.721} C_VEL
LIN {X 0,Y 591.984,Z 95.745,A -85,B 0,C 180,E1 28317.285,E2 28317.285} C_VEL
LIN {X 0,Y 592.037,Z 95.74,A -85,B 0,C 180,E1 28314.159,E2 28314.159} C_VEL
LIN {X 0,Y 591.976,Z 95.74,A -85,B 0,C 180,E1 28311.075,E2 28311.075} C_VEL
LIN {X 0,Y 592.034,Z 95.742,A -85,B 0,C 180,E1 28307.995,E2 28307.995} C_VEL
LIN {X 0,Y 591.979,Z 95.74,A -85,B 0,C 180,E1 28304.911,E2 28304.911} C_VEL
LIN {X 0,Y 592.003,Z 95.742,A -85,B 0,C 180,E1 28301.712,E2 28301.712} C_VEL
LIN {X 0,Y 591.994,Z 95.735,A -85,B 0,C 180,E1 28298.676,E2 28298.676} C_VEL
LIN {X 0,Y 591.975,Z 95.741,A -85,B 0,C 180,E1 28295.404,E2 28295.404} C_VEL
LIN {X 0,Y 592.028,Z 95.738,A -85,B 0,C 180,E1 28292.369,E2 28292.369} C_VEL
LIN {X 0,Y 591.97,Z 95.74,A -85,B 0,C 180,E1 28289.218,E2 28289.218} C_VEL
LIN {X 0,Y 592.038,Z 95.743,A -85,B 0,C 180,E1 28286.154,E2 28286.154} C_VEL
LIN {X 0,Y 591.973,Z 95.739,A -85,B 0,C 180,E1 28283.07,E2 28283.07} C_VEL
LIN {X 0,Y 591.993,Z 95.74,A -85,B 0,C 180,E1 28279.824,E2 28279.824} C_VEL
LIN {X 0,Y 591.983,Z 95.74,A -85,B 0,C 180,E1 28276.888,E2 28276.888} C_VEL
LIN {X 0,Y 591.977,Z 95.739,A -85,B 0,C 180,E1 28273.678,E2 28273.678} C_VEL
LIN {X 0,Y 592.002,Z 95.74,A -85,B 0,C 180,E1 28270.707,E2 28270.707} C_VEL
LIN {X 0,Y 591.969,Z 95.739,A -85,B 0,C 180,E1 28267.57,E2 28267.57} C_VEL
LIN {X 0,Y 592.026,Z 95.74,A -85,B 0,C 180,E1 28264.553,E2 28264.553} C_VEL
LIN {X 0,Y 591.963,Z 95.739,A -85,B 0,C 180,E1 28261.452,E2 28261.452} C_VEL
LIN {X 0,Y 592.031,Z 95.744,A -85,B 0,C 180,E1 28258.355,E2 28258.355} C_VEL
LIN {X 0,Y 591.962,Z 95.74,A -85,B 0,C 180,E1 28255.349,E2 28255.349} C_VEL
LIN {X 0,Y 592.011,Z 95.743,A -85,B 0,C 180,E1 28252.235,E2 28252.235} C_VEL
LIN {X 0,Y 591.994,Z 95.741,A -85,B 0,C 180,E1 28250.113,E2 28250.113} C_VEL
LIN {X 0,Y 590.946,Z 95.87,A -85,B 0,C 180,E1 28249.367,E2 28249.367} C_VEL
LIN {X 0,Y 584.556,Z 96.665,A -85,B 0,C 180,E1 28247.275,E2 28247.275} C_VEL
LIN {X 0,Y 584.077,Z 96.728,A -85,B 0,C 180,E1 28246.731,E2 28246.731} C_VEL
LIN {X 0,Y 584.02,Z 96.73,A -85,B 0,C 180,E1 28243.591,E2 28243.591} C_VEL
LIN {X 0,Y 584.089,Z 96.732,A -85,B 0,C 180,E1 28240.5,E2 28240.5} C_VEL
LIN {X 0,Y 584.021,Z 96.729,A -85,B 0,C 180,E1 28237.449,E2 28237.449} C_VEL
LIN {X 0,Y 584.051,Z 96.731,A -85,B 0,C 180,E1 28234.219,E2 28234.219} C_VEL
LIN {X 0,Y 584.031,Z 96.728,A -85,B 0,C 180,E1 28231.226,E2 28231.226} C_VEL
LIN {X 0,Y 584.023,Z 96.73,A -85,B 0,C 180,E1 28227.934,E2 28227.934} C_VEL
LIN {X 0,Y 584.069,Z 96.731,A -85,B 0,C 180,E1 28224.887,E2 28224.887} C_VEL
LIN {X 0,Y 584.015,Z 96.732,A -85,B 0,C 180,E1 28221.701,E2 28221.701} C_VEL
LIN {X 0,Y 584.077,Z 96.732,A -85,B 0,C 180,E1 28218.571,E2 28218.571} C_VEL
LIN {X 0,Y 584.016,Z 96.731,A -85,B 0,C 180,E1 28215.554,E2 28215.554} C_VEL
LIN {X 0,Y 584.039,Z 96.733,A -85,B 0,C 180,E1 28212.305,E2 28212.305} C_VEL
LIN {X 0,Y 584.026,Z 96.732,A -85,B 0,C 180,E1 28209.43,E2 28209.43} C_VEL
LIN {X 0,Y 584.021,Z 96.732,A -85,B 0,C 180,E1 28206.081,E2 28206.081} C_VEL
LIN {X 0,Y 584.079,Z 96.733,A -85,B 0,C 180,E1 28202.981,E2 28202.981} C_VEL
LIN {X 0,Y 584.017,Z 96.736,A -85,B 0,C 180,E1 28199.88,E2 28199.88} C_VEL
LIN {X 0,Y 584.035,Z 96.745,A -85,B 0,C 180,E1 28199.428,E2 28199.428} C_VEL
LIN {X 0,Y 585.829,Z 102.851,A -85,B 0,C 180,E1 28198.825,E2 28198.825} C_VEL
LIN {X 0,Y 585.438,Z 140.978,A -85,B 0,C 180,E1 28195.817,E2 28195.817} C_VEL
LIN {X 0,Y 585.196,Z 175.752,A -85,B 0,C 180,E1 28193.187,E2 28193.187} C_VEL
LIN {X 0,Y 585.709,Z 181.11,A -85,B 0,C 180,E1 28193.096,E2 28193.096} C_VEL
LIN {X 0,Y 585.335,Z 384.396,A -85,B 0,C 180,E1 28190.452,E2 28190.452} C_VEL
LIN {X 0,Y 585.221,Z 403.389,A -85,B 0,C 180,E1 28190.016,E2 28190.016} C_VEL
LIN {X 0,Y 585.08,Z 421.72,A -85,B 0,C 180,E1 28189.408,E2 28189.408} C_VEL
LIN {X 0,Y 584.911,Z 439.19,A -85,B 0,C 180,E1 28188.642,E2 28188.642} C_VEL
LIN {X 0,Y 584.744,Z 455.891,A -85,B 0,C 180,E1 28187.719,E2 28187.719} C_VEL
LIN {X 0,Y 584.568,Z 471.723,A -85,B 0,C 180,E1 28186.648,E2 28186.648} C_VEL
LIN {X 0,Y 584.401,Z 486.603,A -85,B 0,C 180,E1 28185.431,E2 28185.431} C_VEL
LIN {X 0,Y 584.248,Z 500.54,A -85,B 0,C 180,E1 28184.064,E2 28184.064} C_VEL
LIN {X 0,Y 584.127,Z 513.345,A -85,B 0,C 180,E1 28182.555,E2 28182.555} C_VEL
LIN {X 0,Y 584.044,Z 524.585,A -85,B 0,C 180,E1 28180.954,E2 28180.954} C_VEL
LIN {X 0,Y 583.977,Z 534.28,A -85,B 0,C 180,E1 28179.261,E2 28179.261} C_VEL
LIN {X 0,Y 583.945,Z 542.219,A -85,B 0,C 180,E1 28177.521,E2 28177.521} C_VEL
LIN {X 0,Y 583.922,Z 548.276,A -85,B 0,C 180,E1 28175.798,E2 28175.798} C_VEL
LIN {X 0,Y 583.918,Z 552.783,A -85,B 0,C 180,E1 28174.025,E2 28174.025} C_VEL
LIN {X 0,Y 583.916,Z 555.739,A -85,B 0,C 180,E1 28172.158,E2 28172.158} C_VEL
LIN {X 0,Y 583.909,Z 556.93,A -85,B 0,C 180,E1 28170.294,E2 28170.294} C_VEL
LIN {X 0,Y 583.915,Z 556.38,A -85,B 0,C 180,E1 28168.429,E2 28168.429} C_VEL
LIN {X 0,Y 583.907,Z 554.078,A -85,B 0,C 180,E1 28166.563,E2 28166.563} C_VEL
LIN {X 0,Y 583.918,Z 550.212,A -85,B 0,C 180,E1 28164.792,E2 28164.792} C_VEL
LIN {X 0,Y 583.935,Z 544.625,A -85,B 0,C 180,E1 28163.017,E2 28163.017} C_VEL
LIN {X 0,Y 583.957,Z 537.631,A -85,B 0,C 180,E1 28161.333,E2 28161.333} C_VEL
LIN {X 0,Y 584.013,Z 528.769,A -85,B 0,C 180,E1 28159.643,E2 28159.643} C_VEL
LIN {X 0,Y 584.086,Z 518.46,A -85,B 0,C 180,E1 28158.045,E2 28158.045} C_VEL
LIN {X 0,Y 584.19,Z 506.722,A -85,B 0,C 180,E1 28156.539,E2 28156.539} C_VEL
LIN {X 0,Y 584.324,Z 493.529,A -85,B 0,C 180,E1 28155.127,E2 28155.127} C_VEL
LIN {X 0,Y 584.492,Z 478.757,A -85,B 0,C 180,E1 28153.809,E2 28153.809} C_VEL
LIN {X 0,Y 584.673,Z 462.892,A -85,B 0,C 180,E1 28152.637,E2 28152.637} C_VEL
LIN {X 0,Y 584.857,Z 445.9,A -85,B 0,C 180,E1 28151.613,E2 28151.613} C_VEL
LIN {X 0,Y 585.026,Z 428.892,A -85,B 0,C 180,E1 28150.791,E2 28150.791} C_VEL
LIN {X 0,Y 585.185,Z 410.239,A -85,B 0,C 180,E1 28150.099,E2 28150.099} C_VEL
LIN {X 0,Y 585.302,Z 391.562,A -85,B 0,C 180,E1 28149.601,E2 28149.601} C_VEL
LIN {X 0,Y 585.375,Z 371.784,A -85,B 0,C 180,E1 28149.271,E2 28149.271} C_VEL
LIN {X 0,Y 585.597,Z 178.07,A -85,B 0,C 180,E1 28146.77,E2 28146.77} C_VEL
LIN {X 0,Y 585.146,Z 175.108,A -85,B 0,C 180,E1 28146.698,E2 28146.698} C_VEL
LIN {X 0,Y 585.458,Z 133.281,A -85,B 0,C 180,E1 28143.496,E2 28143.496} C_VEL
LIN {X 0,Y 585.846,Z 102.27,A -85,B 0,C 180,E1 28141.035,E2 28141.035} C_VEL
LIN {X 0,Y 584.03,Z 96.736,A -85,B 0,C 180,E1 28140.458,E2 28140.458} C_VEL
LIN {X 0,Y 584.09,Z 96.733,A -85,B 0,C 180,E1 28137.369,E2 28137.369} C_VEL
LIN {X 0,Y 584.039,Z 96.731,A -85,B 0,C 180,E1 28134.241,E2 28134.241} C_VEL
LIN {X 0,Y 584.077,Z 96.721,A -85,B 0,C 180,E1 28131.004,E2 28131.004} C_VEL
LIN {X 0,Y 584.094,Z 96.733,A -85,B 0,C 180,E1 28127.835,E2 28127.835} C_VEL
LIN {X 0,Y 584.07,Z 96.728,A -85,B 0,C 180,E1 28124.578,E2 28124.578} C_VEL
LIN {X 0,Y 584.098,Z 96.723,A -85,B 0,C 180,E1 28121.281,E2 28121.281} C_VEL
LIN {X 0,Y 584.087,Z 96.729,A -85,B 0,C 180,E1 28118.044,E2 28118.044} C_VEL
LIN {X 0,Y 584.091,Z 96.73,A -85,B 0,C 180,E1 28114.747,E2 28114.747} C_VEL
LIN {X 0,Y 584.088,Z 96.726,A -85,B 0,C 180,E1 28111.474,E2 28111.474} C_VEL
LIN {X 0,Y 584.102,Z 96.764,A -85,B 0,C 180,E1 28109.313,E2 28109.313} C_VEL
LIN {X 0,Y 585.679,Z 102.746,A -85,B 0,C 180,E1 28108.779,E2 28108.779} C_VEL
LIN {X 0,Y 585.425,Z 142.367,A -85,B 0,C 180,E1 28105.71,E2 28105.71} C_VEL
LIN {X 0,Y 585.162,Z 175.805,A -85,B 0,C 180,E1 28103.188,E2 28103.188} C_VEL
LIN {X 0,Y 585.681,Z 181.256,A -85,B 0,C 180,E1 28103.095,E2 28103.095} C_VEL
LIN {X 0,Y 585.339,Z 384.438,A -85,B 0,C 180,E1 28100.451,E2 28100.451} C_VEL
LIN {X 0,Y 585.218,Z 403.411,A -85,B 0,C 180,E1 28100.013,E2 28100.013} C_VEL
LIN {X 0,Y 585.073,Z 421.684,A -85,B 0,C 180,E1 28099.409,E2 28099.409} C_VEL
LIN {X 0,Y 584.913,Z 439.193,A -85,B 0,C 180,E1 28098.643,E2 28098.643} C_VEL
LIN {X 0,Y 584.727,Z 456.671,A -85,B 0,C 180,E1 28097.669,E2 28097.669} C_VEL
LIN {X 0,Y 584.559,Z 472.391,A -85,B 0,C 180,E1 28096.598,E2 28096.598} C_VEL
LIN {X 0,Y 584.389,Z 487.166,A -85,B 0,C 180,E1 28095.379,E2 28095.379} C_VEL
LIN {X 0,Y 584.239,Z 501.481,A -85,B 0,C 180,E1 28093.964,E2 28093.964} C_VEL
LIN {X 0,Y 584.129,Z 513.316,A -85,B 0,C 180,E1 28092.556,E2 28092.556} C_VEL
LIN {X 0,Y 584.045,Z 524.595,A -85,B 0,C 180,E1 28090.955,E2 28090.955} C_VEL
LIN {X 0,Y 583.977,Z 534.264,A -85,B 0,C 180,E1 28089.262,E2 28089.262} C_VEL
LIN {X 0,Y 583.945,Z 542.235,A -85,B 0,C 180,E1 28087.521,E2 28087.521} C_VEL
LIN {X 0,Y 583.917,Z 548.271,A -85,B 0,C 180,E1 28085.799,E2 28085.799} C_VEL
LIN {X 0,Y 583.913,Z 552.791,A -85,B 0,C 180,E1 28084.026,E2 28084.026} C_VEL
LIN {X 0,Y 583.912,Z 555.741,A -85,B 0,C 180,E1 28082.159,E2 28082.159} C_VEL
LIN {X 0,Y 583.913,Z 556.934,A -85,B 0,C 180,E1 28080.295,E2 28080.295} C_VEL
LIN {X 0,Y 583.911,Z 556.321,A -85,B 0,C 180,E1 28078.332,E2 28078.332} C_VEL
LIN {X 0,Y 583.917,Z 553.914,A -85,B 0,C 180,E1 28076.466,E2 28076.466} C_VEL
LIN {X 0,Y 583.921,Z 549.704,A -85,B 0,C 180,E1 28074.596,E2 28074.596} C_VEL
LIN {X 0,Y 583.936,Z 543.91,A -85,B 0,C 180,E1 28072.82,E2 28072.82} C_VEL
LIN {X 0,Y 583.969,Z 536.244,A -85,B 0,C 180,E1 28071.037,E2 28071.037} C_VEL
LIN {X 0,Y 584.028,Z 527.018,A -85,B 0,C 180,E1 28069.345,E2 28069.345} C_VEL
LIN {X 0,Y 584.113,Z 516.314,A -85,B 0,C 180,E1 28067.746,E2 28067.746} C_VEL
LIN {X 0,Y 584.224,Z 504.127,A -85,B 0,C 180,E1 28066.238,E2 28066.238} C_VEL
LIN {X 0,Y 584.361,Z 490.111,A -85,B 0,C 180,E1 28064.802,E2 28064.802} C_VEL
LIN {X 0,Y 584.521,Z 475.56,A -85,B 0,C 180,E1 28063.555,E2 28063.555} C_VEL
LIN {X 0,Y 584.699,Z 458.899,A -85,B 0,C 180,E1 28062.382,E2 28062.382} C_VEL
LIN {X 0,Y 584.882,Z 441.976,A -85,B 0,C 180,E1 28061.408,E2 28061.408} C_VEL
LIN {X 0,Y 585.045,Z 424.873,A -85,B 0,C 180,E1 28060.629,E2 28060.629} C_VEL
LIN {X 0,Y 585.203,Z 405.426,A -85,B 0,C 180,E1 28059.954,E2 28059.954} C_VEL
LIN {X 0,Y 585.324,Z 386.681,A -85,B 0,C 180,E1 28059.502,E2 28059.502} C_VEL
LIN {X 0,Y 585.409,Z 355.421,A -85,B 0,C 180,E1 28059.062,E2 28059.062} C_VEL
LIN {X 0,Y 585.562,Z 177.773,A -85,B 0,C 180,E1 28056.765,E2 28056.765} C_VEL
LIN {X 0,Y 585.141,Z 175.119,A -85,B 0,C 180,E1 28056.698,E2 28056.698} C_VEL
LIN {X 0,Y 585.477,Z 134.411,A -85,B 0,C 180,E1 28053.585,E2 28053.585} C_VEL
LIN {X 0,Y 585.504,Z 101.73,A -85,B 0,C 180,E1 28051.101,E2 28051.101} C_VEL
LIN {X 0,Y 584.069,Z 96.732,A -85,B 0,C 180,E1 28050.686,E2 28050.686} C_VEL
LIN {X 0,Y 584.1,Z 96.729,A -85,B 0,C 180,E1 28047.486,E2 28047.486} C_VEL
LIN {X 0,Y 584.048,Z 96.729,A -85,B 0,C 180,E1 28044.405,E2 28044.405} C_VEL
LIN {X 0,Y 584.07,Z 96.732,A -85,B 0,C 180,E1 28041.161,E2 28041.161} C_VEL
LIN {X 0,Y 584.055,Z 96.73,A -85,B 0,C 180,E1 28038.114,E2 28038.114} C_VEL
LIN {X 0,Y 584.029,Z 96.732,A -85,B 0,C 180,E1 28034.858,E2 28034.858} C_VEL
LIN {X 0,Y 584.089,Z 96.732,A -85,B 0,C 180,E1 28031.725,E2 28031.725} C_VEL
LIN {X 0,Y 584.023,Z 96.733,A -85,B 0,C 180,E1 28028.674,E2 28028.674} C_VEL
LIN {X 0,Y 584.059,Z 96.732,A -85,B 0,C 180,E1 28025.475,E2 28025.475} C_VEL
LIN {X 0,Y 584.055,Z 96.86,A -85,B 0,C 180,E1 28023.117,E2 28023.117} C_VEL
LIN {X 0,Y 586.632,Z 103.839,A -85,B 0,C 180,E1 28022.503,E2 28022.503} C_VEL
LIN {X 0,Y 586.177,Z 152.105,A -85,B 0,C 180,E1 28019.479,E2 28019.479} C_VEL
LIN {X 0,Y 586.19,Z 163.538,A -85,B 0,C 180,E1 28018.801,E2 28018.801} C_VEL
